KUKA KRL program: MyProgram_227().src

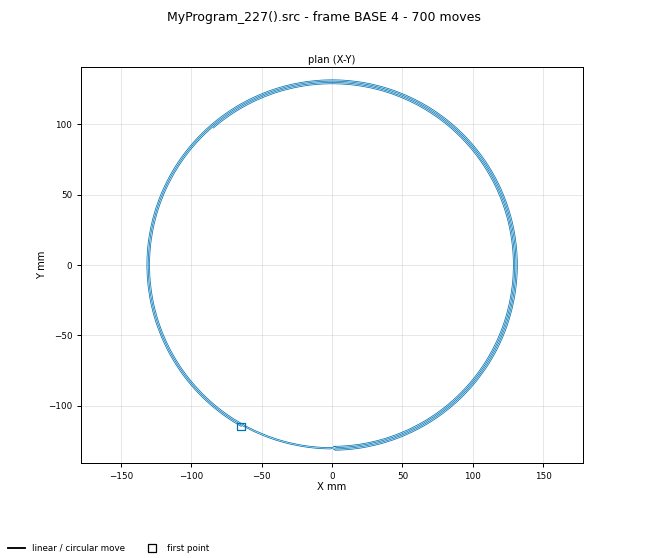
[picture p0: tool path of MyProgram_227().src in frame BASE 4, 700 of 700 moves have a stored position in this frame; points joined in program order, loops and branches not executed]
&ACCESS RVP
&REL 1
&PARAM TEMPLATE = C:\KRC\Roboter\Template\vorgabe
&PARAM EDITMASK = *
DEF MyProgram_227()
; ---- Setting reference (Base) ----
$BASE = BASE_DATA[4]

; --------------------------
; ---- Setting tool (TCP) ----
$TOOL = TOOL_DATA[3]
; --------------------------

$VEL.CP = VEL_APROX_PRINT
Startdeposition()
$VEL.CP = VEL_PRINT
LIN {X -64.5024,Y -114.7242,Z 156,A -121.3808,B 20.2003,C -0.5364,E1 20.1278,E2 209.4297} C_DIS
LIN {X -69.89,Y -111.5247,Z 156,A -124.1594,B 20.2003,C -0.5384,E1 20.1212,E2 212.2133} C_DIS
LIN {X -73.6579,Y -109.0722,Z 156,A -126.0502,B 20.2001,C -0.5441,E1 20.1168,E2 214.0953} C_DIS
LIN {X -77.2991,Y -106.5226,Z 156,A -128.0102,B 20.2001,C -0.5464,E1 20.1123,E2 216.0574} C_DIS
LIN {X -80.7887,Y -103.9011,Z 156,A -129.8858,B 20.1999,C -0.5507,E1 20.1082,E2 217.9291} C_DIS
LIN {X -84.1988,Y -101.1577,Z 156,A -131.8469,B 20.1999,C -0.552,E1 20.1039,E2 219.8956} C_DIS
LIN {X -87.3975,Y -98.4072,Z 156,A -133.6968,B 20.1998,C -0.555,E1 20.1,E2 221.746} C_DIS
LIN {X -90.6409,Y -95.4285,Z 156,A -135.5086,B 20.1996,C -0.563,E1 20.0963,E2 223.5439} C_DIS
LIN {X -93.5164,Y -92.6117,Z 156,A -137.4058,B 20.1996,C -0.561,E1 20.0926,E2 225.457} C_DIS
LIN {X -96.644,Y -89.3436,Z 156,A -139.4007,B 20.1996,C -0.5643,E1 20.0887,E2 227.4534} C_DIS
LIN {X -99.6561,Y -85.9703,Z 156,A -141.3321,B 20.1994,C -0.5702,E1 20.0852,E2 229.3787} C_DIS
LIN {X -102.7577,Y -82.2386,Z 156,A -143.5047,B 20.1994,C -0.5727,E1 20.0813,E2 231.5566} C_DIS
LIN {X -105.5327,Y -78.6451,Z 156,A -145.4674,B 20.1992,C -0.578,E1 20.078,E2 233.5158} C_DIS
LIN {X -108.1949,Y -74.9409,Z 156,A -147.3614,B 20.1989,C -0.5864,E1 20.075,E2 235.397} C_DIS
LIN {X -112.0608,Y -69.0263,Z 156,A -150.3782,B 20.1987,C -0.5965,E1 20.0705,E2 238.4037} C_DIS
LIN {X -115.078,Y -63.8693,Z 156,A -153.1743,B 20.1987,C -0.5959,E1 20.0665,E2 241.22} C_DIS
LIN {X -117.1648,Y -59.9514,Z 156,A -154.8834,B 20.1983,C -0.6097,E1 20.0643,E2 242.9005} C_DIS
LIN {X -118.6307,Y -56.9959,Z 156,A -157.3435,B 20.1993,C -0.575,E1 20.0612,E2 245.4789} C_DIS
LIN {X -121.1915,Y -51.3301,Z 156,A -159.1211,B 20.1981,C -0.6176,E1 20.0594,E2 247.1447} C_DIS
LIN {X -124.2996,Y -43.2591,Z 156,A -163.0083,B 20.1979,C -0.6237,E1 20.0555,E2 251.0416} C_DIS
LIN {X -125.3813,Y -40.0159,Z 156,A -164.4771,B 20.1977,C -0.6288,E1 20.0542,E2 252.5062} C_DIS
LIN {X -126.4456,Y -36.5168,Z 156,A -166.1537,B 20.1977,C -0.6304,E1 20.0529,E2 254.1906} C_DIS
LIN {X -127.474,Y -32.7456,Z 156,A -167.8537,B 20.1975,C -0.6355,E1 20.0517,E2 255.8881} C_DIS
LIN {X -128.2429,Y -29.5906,Z 156,A -169.2782,B 20.1974,C -0.6394,E1 20.0508,E2 257.3118} C_DIS
LIN {X -128.843,Y -26.8636,Z 156,A -170.5109,B 20.1974,C -0.6424,E1 20.0501,E2 258.5449} C_DIS
LIN {X -129.6876,Y -22.4383,Z 156,A -172.5834,B 20.1973,C -0.6443,E1 20.049,E2 260.6277} C_DIS
LIN {X -130.7797,Y -14.7915,Z 156,A -176.0889,B 20.1971,C -0.6494,E1 20.0477,E2 264.1449} C_DIS
LIN {X -131.3696,Y -7.9913,Z 156,A -178.8053,B 20.1965,C -0.6682,E1 20.0471,E2 266.827} C_DIS
LIN {X -131.6089,Y -1.0846,Z 156,A 178.2982,B 20.1961,C -0.6818,E1 20.0469,E2 269.7058} C_DIS
LIN {X -131.5118,Y 5.1452,Z 156,A 175.3937,B 20.1961,C -0.6831,E1 20.0471,E2 272.6287} C_DIS
LIN {X -131.3238,Y 8.7353,Z 156,A 173.6587,B 20.1961,C -0.6817,E1 20.0474,E2 274.3812} C_DIS
LIN {X -131.0445,Y 12.2177,Z 156,A 171.8386,B 20.1963,C -0.6754,E1 20.0478,E2 276.2337} C_DIS
LIN {X -130.5968,Y 16.3351,Z 156,A 170.3498,B 20.1957,C -0.6927,E1 20.0483,E2 277.6831} C_DIS
LIN {X -130.0557,Y 20.1816,Z 156,A 168.5773,B 20.1957,C -0.695,E1 20.049,E2 279.4623} C_DIS
LIN {X -129.1113,Y 25.5452,Z 156,A 166.2566,B 20.1953,C -0.7043,E1 20.0502,E2 281.7735} C_DIS
LIN {X -128.3484,Y 29.1287,Z 156,A 164.8371,B 20.1949,C -0.7158,E1 20.0511,E2 283.1699} C_DIS
LIN {X -127.6208,Y 32.1674,Z 156,A 163.3923,B 20.1949,C -0.7168,E1 20.052,E2 284.6224} C_DIS
LIN {X -126.7498,Y 35.4433,Z 156,A 161.9281,B 20.1947,C -0.7218,E1 20.0531,E2 286.0828} C_DIS
LIN {X -125.9037,Y 38.3411,Z 156,A 160.6577,B 20.1945,C -0.7275,E1 20.0541,E2 287.3459} C_DIS
LIN {X -124.9623,Y 41.3068,Z 156,A 159.1923,B 20.1945,C -0.7275,E1 20.0554,E2 288.8222} C_DIS
LIN {X -123.8552,Y 44.5154,Z 156,A 157.764,B 20.1943,C -0.7338,E1 20.0567,E2 290.2423} C_DIS
LIN {X -122.7696,Y 47.4281,Z 156,A 156.44,B 20.1941,C -0.7389,E1 20.058,E2 291.5607} C_DIS
LIN {X -121.5158,Y 50.5536,Z 156,A 154.8555,B 20.1941,C -0.7389,E1 20.0597,E2 293.1566} C_DIS
LIN {X -119.7827,Y 54.538,Z 156,A 152.3207,B 20.1948,C -0.7204,E1 20.0627,E2 295.763} C_DIS
LIN {X -117.5878,Y 59.1205,Z 156,A 150.668,B 20.1938,C -0.7476,E1 20.0646,E2 297.3475} C_DIS
LIN {X -115.5845,Y 62.9479,Z 156,A 148.762,B 20.1937,C -0.752,E1 20.0671,E2 299.2535} C_DIS
LIN {X -113.2985,Y 66.9761,Z 156,A 146.8963,B 20.1933,C -0.7634,E1 20.0697,E2 301.0984} C_DIS
LIN {X -111.4896,Y 69.9457,Z 156,A 145.2337,B 20.1933,C -0.7619,E1 20.0722,E2 302.7761} C_DIS
LIN {X -109.3086,Y 73.307,Z 156,A 143.4515,B 20.1933,C -0.7652,E1 20.0749,E2 304.5598} C_DIS
LIN {X -106.8382,Y 76.8632,Z 156,A 141.5225,B 20.1931,C -0.7686,E1 20.078,E2 306.4911} C_DIS
LIN {X -104.1297,Y 80.4938,Z 156,A 139.5695,B 20.1929,C -0.7744,E1 20.0813,E2 308.4389} C_DIS
LIN {X -101.2648,Y 84.0694,Z 156,A 137.5744,B 20.1927,C -0.7795,E1 20.0848,E2 310.4311} C_DIS
LIN {X -98.3299,Y 87.485,Z 156,A 135.5579,B 20.1926,C -0.7822,E1 20.0886,E2 312.4512} C_DIS
LIN {X -95.3804,Y 90.6912,Z 156,A 133.6485,B 20.1924,C -0.7863,E1 20.0922,E2 314.3593} C_DIS
LIN {X -92.0975,Y 94.0227,Z 156,A 131.6693,B 20.1922,C -0.7932,E1 20.0961,E2 316.3289} C_DIS
LIN {X -89.054,Y 96.9102,Z 156,A 129.8341,B 20.192,C -0.797,E1 20.0998,E2 318.1626} C_DIS
LIN {X -85.7986,Y 99.8039,Z 156,A 127.9139,B 20.192,C -0.8002,E1 20.1039,E2 320.083} C_DIS
LIN {X -82.5599,Y 102.4991,Z 156,A 126.0958,B 20.1917,C -0.8047,E1 20.1078,E2 321.8967} C_DIS
LIN {X -79.2878,Y 105.0507,Z 156,A 124.262,B 20.1917,C -0.8073,E1 20.1118,E2 323.7313} C_DIS
LIN {X -75.7971,Y 107.5965,Z 156,A 122.3591,B 20.1915,C -0.8102,E1 20.1162,E2 325.6344} C_DIS
LIN {X -72.1164,Y 110.0978,Z 156,A 120.4059,B 20.1915,C -0.8132,E1 20.1207,E2 327.5869} C_DIS
LIN {X -68.5529,Y 112.3513,Z 156,A 118.5367,B 20.1913,C -0.8152,E1 20.1251,E2 329.4578} C_DIS
LIN {X -64.9667,Y 114.4623,Z 156,A 116.7463,B 20.1912,C -0.8191,E1 20.1294,E2 331.2435} C_DIS
LIN {X -61.8178,Y 116.1928,Z 156,A 114.9516,B 20.1914,C -0.8127,E1 20.1339,E2 333.0633} C_DIS
LIN {X -58.9034,Y 117.6973,Z 156,A 113.719,B 20.1911,C -0.8225,E1 20.1369,E2 334.2716} C_DIS
LIN {X -55.5927,Y 119.295,Z 156,A 112.0742,B 20.1911,C -0.8231,E1 20.1411,E2 335.9197} C_DIS
LIN {X -49.197,Y 122.0712,Z 156,A 109.1849,B 20.1906,C -0.833,E1 20.1485,E2 338.7888} C_DIS
LIN {X -45.7308,Y 123.4124,Z 156,A 107.5441,B 20.1906,C -0.8341,E1 20.1528,E2 340.4307} C_DIS
LIN {X -42.1881,Y 124.6688,Z 156,A 105.8112,B 20.1906,C -0.8322,E1 20.1574,E2 342.1733} C_DIS
LIN {X -38.1859,Y 125.9512,Z 156,A 103.9702,B 20.1906,C -0.8338,E1 20.1623,E2 344.0139} C_DIS
LIN {X -33.5783,Y 127.2571,Z 156,A 101.5534,B 20.191,C -0.8227,E1 20.1689,E2 346.4674} C_DIS
LIN {X -29.7777,Y 128.2002,Z 156,A 100.0213,B 20.1907,C -0.831,E1 20.173,E2 347.9782} C_DIS
LIN {X -26.3077,Y 128.9561,Z 156,A 98.0483,B 20.1913,C -0.8153,E1 20.1785,E2 349.9994} C_DIS
LIN {X -21.1994,Y 129.8945,Z 156,A 96.3348,B 20.1904,C -0.8385,E1 20.1831,E2 351.6477} C_DIS
LIN {X -17.142,Y 130.4912,Z 156,A 94.7251,B 20.1901,C -0.8466,E1 20.1874,E2 353.2356} C_DIS
LIN {X -10.1792,Y 131.2195,Z 156,A 91.5234,B 20.1903,C -0.8417,E1 20.1964,E2 356.4535} C_DIS
LIN {X -6.3873,Y 131.4575,Z 156,A 89.89,B 20.1903,C -0.8431,E1 20.2009,E2 358.0836} C_DIS
LIN {X -2.1877,Y 131.5943,Z 156,A 88.078,B 20.1902,C -0.8442,E1 20.206,E2 359.8925} C_DIS
LIN {X 1.9611,Y 131.5981,Z 156,A 86.5669,B 20.1897,C -0.8564,E1 20.2101,E2 361.3682} C_DIS
LIN {X 5.8923,Y 131.4824,Z 156,A 84.5148,B 20.1903,C -0.8426,E1 20.2159,E2 363.4595} C_DIS
LIN {X 9.6611,Y 131.2574,Z 156,A 82.9336,B 20.1902,C -0.8451,E1 20.2203,E2 365.0327} C_DIS
LIN {X 13.7775,Y 130.8896,Z 156,A 81.0592,B 20.1902,C -0.8418,E1 20.2256,E2 366.9154} C_DIS
LIN {X 19.5443,Y 130.1544,Z 156,A 78.571,B 20.1902,C -0.8428,E1 20.2324,E2 369.3978} C_DIS
LIN {X 23.245,Y 129.5433,Z 156,A 76.9573,B 20.1902,C -0.843,E1 20.2369,E2 371.0089} C_DIS
LIN {X 28.1767,Y 128.5613,Z 156,A 74.7152,B 20.1904,C -0.8397,E1 20.243,E2 373.2569} C_DIS
LIN {X 32.0967,Y 127.6387,Z 156,A 73.1025,B 20.1902,C -0.8444,E1 20.2473,E2 374.8529} C_DIS
LIN {X 35.2064,Y 126.8161,Z 156,A 71.485,B 20.1906,C -0.8345,E1 20.2518,E2 376.4958} C_DIS
LIN {X 39.8423,Y 125.4367,Z 156,A 69.5312,B 20.1904,C -0.8392,E1 20.2569,E2 378.4316} C_DIS
LIN {X 43.2726,Y 124.2949,Z 156,A 68.0856,B 20.1902,C -0.8431,E1 20.2607,E2 379.8622} C_DIS
LIN {X 49.0275,Y 122.1395,Z 156,A 65.3591,B 20.1904,C -0.8384,E1 20.2679,E2 382.595} C_DIS
LIN {X 52.1568,Y 120.8362,Z 156,A 63.8884,B 20.1904,C -0.837,E1 20.2716,E2 384.0654} C_DIS
LIN {X 55.0772,Y 119.5334,Z 156,A 62.6797,B 20.1902,C -0.8431,E1 20.2746,E2 385.2526} C_DIS
LIN {X 57.4891,Y 118.395,Z 156,A 61.1776,B 20.1909,C -0.8272,E1 20.2785,E2 386.7954} C_DIS
LIN {X 61.0133,Y 116.6152,Z 156,A 59.6562,B 20.1906,C -0.8333,E1 20.2823,E2 388.2938} C_DIS
LIN {X 63.6126,Y 115.2201,Z 156,A 58.0731,B 20.1912,C -0.8189,E1 20.2862,E2 389.9127} C_DIS
LIN {X 68.2018,Y 112.5644,Z 156,A 55.9412,B 20.191,C -0.823,E1 20.2913,E2 392.0246} C_DIS
LIN {X 71.9413,Y 110.2124,Z 156,A 54.0685,B 20.191,C -0.8221,E1 20.2957,E2 393.8921} C_DIS
LIN {X 75.4654,Y 107.83,Z 156,A 52.1497,B 20.1913,C -0.8162,E1 20.3001,E2 395.8197} C_DIS
LIN {X 78.7314,Y 105.4685,Z 156,A 50.4574,B 20.1913,C -0.8158,E1 20.3039,E2 397.5056} C_DIS
LIN {X 82.2037,Y 102.7855,Z 156,A 48.5796,B 20.1913,C -0.8137,E1 20.308,E2 399.3806} C_DIS
LIN {X 85.4731,Y 100.0832,Z 156,A 46.7923,B 20.1914,C -0.8127,E1 20.3119,E2 401.162} C_DIS
LIN {X 88.738,Y 97.1994,Z 156,A 44.5515,B 20.1921,C -0.7942,E1 20.3166,E2 403.4449} C_DIS
LIN {X 91.3003,Y 94.7976,Z 156,A 43.2428,B 20.1919,C -0.8004,E1 20.3192,E2 404.7286} C_DIS
LIN {X 94.5144,Y 91.5928,Z 156,A 41.319,B 20.1919,C -0.7985,E1 20.3229,E2 406.6478} C_DIS
LIN {X 97.1681,Y 88.7731,Z 156,A 39.6028,B 20.1922,C -0.7934,E1 20.3262,E2 408.3689} C_DIS
LIN {X 99.6795,Y 85.9431,Z 156,A 37.9873,B 20.1922,C -0.7911,E1 20.3292,E2 409.982} C_DIS
LIN {X 102.9297,Y 82.0225,Z 156,A 35.8142,B 20.1924,C -0.7878,E1 20.333,E2 412.1518} C_DIS
LIN {X 105.4685,Y 78.7314,Z 156,A 34.1292,B 20.1924,C -0.7888,E1 20.3358,E2 413.8237} C_DIS
LIN {X 108.7981,Y 74.0628,Z 156,A 31.5163,B 20.1928,C -0.7775,E1 20.3401,E2 416.453} C_DIS
LIN {X 111.0812,Y 70.5928,Z 156,A 29.6889,B 20.193,C -0.772,E1 20.3428,E2 418.2846} C_DIS
LIN {X 113.4512,Y 66.7161,Z 156,A 27.7613,B 20.193,C -0.7691,E1 20.3456,E2 420.2082} C_DIS
LIN {X 115.67,Y 62.7911,Z 156,A 26.0407,B 20.1929,C -0.7744,E1 20.3479,E2 421.9021} C_DIS
LIN {X 118.0921,Y 58.1031,Z 156,A 23.5923,B 20.1933,C -0.7615,E1 20.351,E2 424.3711} C_DIS
LIN {X 119.7335,Y 54.6444,Z 156,A 21.83,B 20.1937,C -0.7526,E1 20.3531,E2 426.1469} C_DIS
LIN {X 121.347,Y 50.9576,Z 156,A 20.2893,B 20.1935,C -0.757,E1 20.3548,E2 427.6645} C_DIS
LIN {X 122.5599,Y 47.9675,Z 156,A 18.9069,B 20.1936,C -0.7539,E1 20.3562,E2 429.046} C_DIS
LIN {X 123.6574,Y 45.0642,Z 156,A 17.4929,B 20.1939,C -0.7472,E1 20.3576,E2 430.4693} C_DIS
LIN {X 124.7234,Y 42.0241,Z 156,A 16.1047,B 20.1939,C -0.7437,E1 20.3589,E2 431.8576} C_DIS
LIN {X 125.5276,Y 39.558,Z 156,A 14.9124,B 20.1942,C -0.7376,E1 20.3599,E2 433.059} C_DIS
LIN {X 126.8788,Y 34.9821,Z 156,A 13.0111,B 20.1942,C -0.7392,E1 20.3614,E2 434.9419} C_DIS
LIN {X 127.8142,Y 31.3943,Z 156,A 10.8889,B 20.1951,C -0.7119,E1 20.3628,E2 437.1271} C_DIS
LIN {X 128.6714,Y 27.6669,Z 156,A 9.2288,B 20.1952,C -0.707,E1 20.3638,E2 438.789} C_DIS
LIN {X 129.4575,Y 23.724,Z 156,A 7.8543,B 20.1949,C -0.7182,E1 20.3645,E2 440.1211} C_DIS
LIN {X 130.0535,Y 20.1963,Z 156,A 6.3721,B 20.1949,C -0.7168,E1 20.3652,E2 441.5965} C_DIS
LIN {X 130.8383,Y 14.2538,Z 156,A 3.5714,B 20.1955,C -0.7002,E1 20.3661,E2 444.424} C_DIS
LIN {X 131.2658,Y 9.5455,Z 156,A 1.7609,B 20.1953,C -0.7047,E1 20.3665,E2 446.2078} C_DIS
LIN {X 131.4776,Y 5.9883,Z 156,A 0.1341,B 20.1956,C -0.6965,E1 20.3668,E2 447.8461} C_DIS
LIN {X 131.5938,Y 2.2195,Z 156,A -1.4535,B 20.1956,C -0.6937,E1 20.3668,E2 449.4297} C_DIS
LIN {X 131.5982,Y -1.9522,Z 156,A -3.2301,B 20.1958,C -0.6897,E1 20.3668,E2 451.2044} C_DIS
LIN {X 131.4915,Y -5.6661,Z 156,A -4.9406,B 20.1961,C -0.6805,E1 20.3667,E2 452.9287} C_DIS
LIN {X 131.2776,Y -9.3838,Z 156,A -6.319,B 20.1959,C -0.6862,E1 20.3664,E2 454.2803} C_DIS
LIN {X 130.6782,Y -15.6533,Z 156,A -9.1651,B 20.1964,C -0.6728,E1 20.3656,E2 457.1434} C_DIS
LIN {X 130.144,Y -19.6118,Z 156,A -10.7532,B 20.1964,C -0.6741,E1 20.365,E2 458.7162} C_DIS
LIN {X 129.3929,Y -24.0765,Z 156,A -12.882,B 20.1967,C -0.6608,E1 20.364,E2 460.8672} C_DIS
LIN {X 127.674,Y -31.9578,Z 156,A -17.4583,B 20.1985,C -0.603,E1 20.361,E2 465.5762} C_DIS
LIN {X 125.5974,Y -39.3394,Z 156,A -19.7302,B 20.1974,C -0.6396,E1 20.3592,E2 467.7264} C_DIS
LIN {X 124.5474,Y -42.5443,Z 156,A -21.0624,B 20.1974,C -0.6412,E1 20.3581,E2 469.0446} C_DIS
LIN {X 123.3126,Y -45.9974,Z 156,A -23.4632,B 20.1985,C -0.6009,E1 20.3556,E2 471.5444} C_DIS
LIN {X 121.1237,Y -51.4912,Z 156,A -25.2866,B 20.1978,C -0.6263,E1 20.3538,E2 473.282} C_DIS
LIN {X 119.6012,Y -54.9305,Z 156,A -26.6816,B 20.1976,C -0.6323,E1 20.3522,E2 474.6503} C_DIS
LIN {X 118.8149,Y -56.6104,Z 156,A -28.0066,B 20.1984,C -0.607,E1 20.3505,E2 476.039} C_DIS
LIN {X 117.2458,Y -59.7924,Z 156,A -29.0782,B 20.1979,C -0.6234,E1 20.3493,E2 477.0561} C_DIS
LIN {X 115.7121,Y -62.7141,Z 156,A -30.7188,B 20.1983,C -0.6102,E1 20.3471,E2 478.7237} C_DIS
LIN {X 113.701,Y -66.2907,Z 156,A -32.4644,B 20.1983,C -0.6069,E1 20.3446,E2 480.4673} C_DIS
LIN {X 111.5286,Y -69.8839,Z 156,A -34.2997,B 20.1985,C -0.6015,E1 20.3419,E2 482.3064} C_DIS
LIN {X 109.1962,Y -73.4747,Z 156,A -36.1344,B 20.1986,C -0.5977,E1 20.3391,E2 484.1405} C_DIS
LIN {X 104.0032,Y -80.6569,Z 156,A -40.1372,B 20.1991,C -0.5811,E1 20.3325,E2 488.1666} C_DIS
LIN {X 101.5007,Y -83.7846,Z 156,A -42.1923,B 20.1996,C -0.563,E1 20.3288,E2 490.2619} C_DIS
LIN {X 98.4389,Y -87.3616,Z 156,A -43.6096,B 20.199,C -0.5856,E1 20.3263,E2 491.6061} C_DIS
LIN {X 93.3518,Y -92.7774,Z 156,A -46.8661,B 20.1992,C -0.5768,E1 20.32,E2 494.8701} C_DIS
LIN {X 88.3975,Y -97.5095,Z 156,A -50.1148,B 20.1997,C -0.5583,E1 20.3133,E2 498.1552} C_DIS
LIN {X 83.9468,Y -101.3663,Z 156,A -52.4094,B 20.1995,C -0.5644,E1 20.3085,E2 500.4208} C_DIS
LIN {X 78.3102,Y -105.7821,Z 156,A -55.623,B 20.1998,C -0.5537,E1 20.3013,E2 503.6504} C_DIS
LIN {X 74.6594,Y -108.3892,Z 156,A -57.5017,B 20.1998,C -0.5531,E1 20.297,E2 505.5226} C_DIS
LIN {X 71.3089,Y -110.6229,Z 156,A -59.4292,B 20.2001,C -0.5422,E1 20.2925,E2 507.4733} C_DIS
LIN {X 66.739,Y -113.4378,Z 156,A -61.5372,B 20.2,C -0.5479,E1 20.2875,E2 509.5566} C_DIS
LIN {X 63.2524,Y -115.4184,Z 156,A -63.1592,B 20.2,C -0.5503,E1 20.2836,E2 511.1658} C_DIS
LIN {X 57.3027,Y -118.4841,Z 156,A -66.1346,B 20.2001,C -0.5429,E1 20.2762,E2 514.1521} C_DIS
LIN {X 53.848,Y -120.0921,Z 156,A -67.7383,B 20.2001,C -0.5429,E1 20.2721,E2 515.7509} C_DIS
LIN {X 51.3763,Y -121.1722,Z 156,A -69.004,B 20.2003,C -0.5372,E1 20.2688,E2 517.0289} C_DIS
LIN {X 47.3272,Y -122.8088,Z 156,A -70.9608,B 20.2003,C -0.5323,E1 20.2637,E2 518.9944} C_DIS
LIN {X 43.1661,Y -124.3319,Z 156,A -72.7643,B 20.2003,C -0.5353,E1 20.259,E2 520.7846} C_DIS
LIN {X 37.2335,Y -126.2358,Z 156,A -75.7877,B 20.2007,C -0.519,E1 20.2508,E2 523.848} C_DIS
LIN {X 34.0665,Y -127.1269,Z 156,A -76.89,B 20.2004,C -0.5316,E1 20.248,E2 524.9119} C_DIS
LIN {X 30.9231,Y -127.9278,Z 156,A -78.2553,B 20.2004,C -0.5322,E1 20.2443,E2 526.2727} C_DIS
LIN {X 24.2335,Y -129.3629,Z 156,A -81.2641,B 20.2004,C -0.5284,E1 20.2361,E2 529.2877} C_DIS
LIN {X 21.8709,Y -129.7825,Z 156,A -82.7006,B 20.2009,C -0.5112,E1 20.232,E2 530.772} C_DIS
LIN {X 18.2798,Y -130.3371,Z 156,A -84.0182,B 20.2007,C -0.5213,E1 20.2284,E2 532.0591} C_DIS
LIN {X 14.3884,Y -130.8238,Z 156,A -85.6588,B 20.2007,C -0.5231,E1 20.2239,E2 533.6928} C_DIS
LIN {X 10.3975,Y -131.2028,Z 156,A -87.4427,B 20.2007,C -0.5206,E1 20.2189,E2 535.4825} C_DIS
LIN {X 6.4754,Y -131.4531,Z 156,A -89.1069,B 20.2007,C -0.522,E1 20.2143,E2 537.142} C_DIS
LIN {X 2.2514,Y -131.5932,Z 156,A -90.9121,B 20.2007,C -0.5229,E1 20.2092,E2 538.944} C_DIS
LIN {X 2.2514,Y -131.5932,Z 156,A -90.9121,B 20.2007,C -0.5229,E1 20.2092,E2 538.944} C_DIS
Enddeposition()
LIN {X 0.9052,Y -130.6755,Z 156,A -91.1331,B 18.9222,C -0.3682,E1 18.9261,E2 539.5117} C_DIS
Startdeposition()
$VEL.CP = VEL_PRINT
LIN {X 5.0067,Y -130.5828,Z 156,A -88.6405,B 18.9216,C -0.3957,E1 18.9333,E2 536.9351} C_DIS
LIN {X 8.8903,Y -130.3774,Z 156,A -86.9352,B 18.9216,C -0.3963,E1 18.9381,E2 535.2288} C_DIS
LIN {X 12.4269,Y -130.0864,Z 156,A -85.3683,B 18.9216,C -0.3975,E1 18.9424,E2 533.6595} C_DIS
LIN {X 16.5957,Y -129.621,Z 156,A -83.5782,B 18.9216,C -0.3965,E1 18.9474,E2 531.8742} C_DIS
LIN {X 22.9346,Y -128.6502,Z 156,A -80.8451,B 18.9216,C -0.3953,E1 18.9549,E2 529.1486} C_DIS
LIN {X 30.7927,Y -126.9988,Z 156,A -77.431,B 18.9216,C -0.3939,E1 18.9642,E2 525.7449} C_DIS
LIN {X 36.1822,Y -125.5707,Z 156,A -74.4087,B 18.9211,C -0.4195,E1 18.9725,E2 522.6506} C_DIS
LIN {X 39.6405,Y -124.521,Z 156,A -73.143,B 18.9214,C -0.4084,E1 18.9758,E2 521.4221} C_DIS
LIN {X 43.8451,Y -123.1043,Z 156,A -71.2127,B 18.9214,C -0.4101,E1 18.9809,E2 519.4919} C_DIS
LIN {X 47.3236,Y -121.8083,Z 156,A -69.6873,B 18.9214,C -0.4081,E1 18.9848,E2 517.9772} C_DIS
LIN {X 49.9928,Y -120.738,Z 156,A -68.221,B 18.9212,C -0.4181,E1 18.9887,E2 516.4847} C_DIS
LIN {X 54.5977,Y -118.7264,Z 156,A -66.431,B 18.9214,C -0.4045,E1 18.9931,E2 514.7424} C_DIS
LIN {X 59.6854,Y -116.2524,Z 156,A -63.7114,B 18.9212,C -0.418,E1 19,E2 511.9913} C_DIS
LIN {X 63.512,Y -114.2085,Z 156,A -61.7575,B 18.921,C -0.4232,E1 19.0048,E2 510.0291} C_DIS
LIN {X 67.1764,Y -112.0924,Z 156,A -59.6628,B 18.9208,C -0.4362,E1 19.01,E2 507.9031} C_DIS
LIN {X 70.0987,Y -110.2888,Z 156,A -58.3792,B 18.9209,C -0.4299,E1 19.0129,E2 506.6447} C_DIS
LIN {X 73.714,Y -107.9056,Z 156,A -56.5242,B 18.9209,C -0.4317,E1 19.0172,E2 504.7926} C_DIS
LIN {X 77.2438,Y -105.4073,Z 156,A -54.895,B 18.921,C -0.4244,E1 19.0208,E2 503.1934} C_DIS
LIN {X 82.5021,Y -101.3447,Z 156,A -51.7147,B 18.9206,C -0.4414,E1 19.0279,E2 499.9771} C_DIS
LIN {X 85.9475,Y -98.4394,Z 156,A -49.7809,B 18.9206,C -0.4439,E1 19.032,E2 498.0458} C_DIS
LIN {X 88.9068,Y -95.775,Z 156,A -47.5299,B 18.92,C -0.4688,E1 19.0368,E2 495.7309} C_DIS
LIN {X 92.363,Y -92.4472,Z 156,A -45.9363,B 18.9204,C -0.4525,E1 19.0398,E2 494.1966} C_DIS
LIN {X 96.4676,Y -88.1557,Z 156,A -43.4115,B 18.9204,C -0.4554,E1 19.0446,E2 491.6777} C_DIS
LIN {X 100.555,Y -83.4625,Z 156,A -40.6492,B 18.9201,C -0.4636,E1 19.0497,E2 488.9074} C_DIS
LIN {X 103.3035,Y -80.0355,Z 156,A -37.9705,B 18.9192,C -0.5001,E1 19.0544,E2 486.134} C_DIS
LIN {X 106.9356,Y -75.1141,Z 156,A -36.0855,B 18.9199,C -0.4736,E1 19.0573,E2 484.3425} C_DIS
LIN {X 109.2436,Y -71.7158,Z 156,A -34.2865,B 18.9198,C -0.4784,E1 19.0601,E2 482.541} C_DIS
LIN {X 111.4646,Y -68.2126,Z 156,A -32.4871,B 18.9197,C -0.4826,E1 19.0627,E2 480.7413} C_DIS
LIN {X 113.7219,Y -64.38,Z 156,A -30.5032,B 18.9195,C -0.4894,E1 19.0655,E2 478.7503} C_DIS
LIN {X 115.7765,Y -60.6019,Z 156,A -28.7571,B 18.9195,C -0.489,E1 19.0678,E2 477.0182} C_DIS
LIN {X 118.4529,Y -55.1891,Z 156,A -26.1109,B 18.9193,C -0.4965,E1 19.071,E2 474.3682} C_DIS
LIN {X 120.2831,Y -51.0789,Z 156,A -23.2694,B 18.9182,C -0.539,E1 19.0743,E2 471.4175} C_DIS
LIN {X 122.6579,Y -45.083,Z 156,A -21.2294,B 18.9189,C -0.514,E1 19.0762,E2 469.4695} C_DIS
LIN {X 123.9393,Y -41.4233,Z 156,A -19.8022,B 18.919,C -0.5077,E1 19.0774,E2 468.0727} C_DIS
LIN {X 124.9991,Y -38.106,Z 156,A -17.4959,B 18.918,C -0.5452,E1 19.0794,E2 465.6693} C_DIS
LIN {X 126.4376,Y -33.0275,Z 156,A -15.7772,B 18.9185,C -0.527,E1 19.0806,E2 464.0197} C_DIS
LIN {X 127.2358,Y -29.8065,Z 156,A -14.0493,B 18.9181,C -0.543,E1 19.0817,E2 462.2564} C_DIS
LIN {X 127.9985,Y -26.3301,Z 156,A -12.8924,B 18.9184,C -0.5308,E1 19.0824,E2 461.146} C_DIS
LIN {X 129.2709,Y -19.1403,Z 156,A -9.6278,B 18.9181,C -0.5434,E1 19.0839,E2 457.8691} C_DIS
LIN {X 130.1332,Y -11.925,Z 156,A -6.6336,B 18.9181,C -0.5452,E1 19.0848,E2 454.8932} C_DIS
LIN {X 130.4338,Y -7.9966,Z 156,A -4.8089,B 18.9178,C -0.5547,E1 19.0852,E2 453.0543} C_DIS
LIN {X 130.6217,Y -3.8656,Z 156,A -3.0252,B 18.9177,C -0.5591,E1 19.0854,E2 451.2714} C_DIS
LIN {X 130.6786,Y -0.3496,Z 156,A -1.4346,B 18.9175,C -0.566,E1 19.0854,E2 449.6726} C_DIS
LIN {X 130.6276,Y 3.6539,Z 156,A 0.2672,B 18.9174,C -0.5692,E1 19.0853,E2 447.9747} C_DIS
LIN {X 130.4451,Y 7.8125,Z 156,A 2.0701,B 18.9172,C -0.5739,E1 19.085,E2 446.1719} C_DIS
LIN {X 130.2398,Y 10.704,Z 156,A 3.7221,B 18.9166,C -0.5939,E1 19.0847,E2 444.4721} C_DIS
LIN {X 129.8527,Y 14.6857,Z 156,A 5.7568,B 18.9161,C -0.6112,E1 19.084,E2 442.4008} C_DIS
LIN {X 129.1444,Y 19.9649,Z 156,A 7.3594,B 18.9168,C -0.5874,E1 19.0834,E2 440.8838} C_DIS
LIN {X 128.7001,Y 22.6556,Z 156,A 8.9728,B 18.9162,C -0.6086,E1 19.0826,E2 439.2184} C_DIS
LIN {X 127.9596,Y 26.5197,Z 156,A 10.3455,B 18.9165,C -0.599,E1 19.0818,E2 437.8859} C_DIS
LIN {X 126.4118,Y 33.1241,Z 156,A 13.1417,B 18.9165,C -0.6004,E1 19.08,E2 435.1073} C_DIS
LIN {X 125.5707,Y 36.1822,Z 156,A 14.4641,B 18.9164,C -0.6017,E1 19.079,E2 433.7913} C_DIS
LIN {X 124.5388,Y 39.5847,Z 156,A 16.1018,B 18.9161,C -0.6096,E1 19.0776,E2 432.1422} C_DIS
LIN {X 123.4248,Y 42.932,Z 156,A 17.6503,B 18.9161,C -0.6141,E1 19.0762,E2 430.5916} C_DIS
LIN {X 122.0893,Y 46.6009,Z 156,A 19.4974,B 18.9157,C -0.6246,E1 19.0744,E2 428.7263} C_DIS
LIN {X 120.6642,Y 50.1697,Z 156,A 21.0297,B 18.9157,C -0.6231,E1 19.0728,E2 427.2102} C_DIS
LIN {X 119.3571,Y 53.2042,Z 156,A 22.4643,B 18.9157,C -0.6265,E1 19.0712,E2 425.7756} C_DIS
LIN {X 118.1494,Y 55.8373,Z 156,A 24.2239,B 18.9148,C -0.6504,E1 19.069,E2 423.9558} C_DIS
LIN {X 116.283,Y 59.6254,Z 156,A 25.6936,B 18.9152,C -0.6395,E1 19.0672,E2 422.5301} C_DIS
LIN {X 114.2241,Y 63.4837,Z 156,A 27.5025,B 18.9152,C -0.6401,E1 19.0648,E2 420.7323} C_DIS
LIN {X 112.2691,Y 66.88,Z 156,A 29.2673,B 18.915,C -0.6465,E1 19.0623,E2 418.9601} C_DIS
LIN {X 109.8864,Y 70.7275,Z 156,A 31.2167,B 18.9148,C -0.6502,E1 19.0594,E2 417.013} C_DIS
LIN {X 106.5969,Y 75.5933,Z 156,A 33.8812,B 18.9145,C -0.6602,E1 19.0552,E2 414.3354} C_DIS
LIN {X 103.5846,Y 79.6721,Z 156,A 36.021,B 18.9145,C -0.6621,E1 19.0516,E2 412.2036} C_DIS
LIN {X 101.568,Y 82.227,Z 156,A 37.6685,B 18.914,C -0.6745,E1 19.0487,E2 410.5286} C_DIS
LIN {X 99.3548,Y 84.8883,Z 156,A 38.9348,B 18.9143,C -0.6677,E1 19.0464,E2 409.2912} C_DIS
LIN {X 96.4696,Y 88.1535,Z 156,A 40.9204,B 18.914,C -0.675,E1 19.0427,E2 407.2952} C_DIS
LIN {X 93.0425,Y 91.7634,Z 156,A 43.0169,B 18.914,C -0.6761,E1 19.0386,E2 405.2073} C_DIS
LIN {X 90.2107,Y 94.548,Z 156,A 45.1123,B 18.9133,C -0.6942,E1 19.0343,E2 403.0684} C_DIS
LIN {X 87.1704,Y 97.3582,Z 156,A 46.5257,B 18.9138,C -0.6814,E1 19.0315,E2 401.702} C_DIS
LIN {X 83.8438,Y 100.2374,Z 156,A 48.1912,B 18.914,C -0.6744,E1 19.028,E2 400.0667} C_DIS
LIN {X 81.1814,Y 102.4057,Z 156,A 49.9517,B 18.9136,C -0.6875,E1 19.0241,E2 398.2751} C_DIS
LIN {X 77.6585,Y 105.1027,Z 156,A 51.8796,B 18.9135,C -0.6902,E1 19.0198,E2 396.3483} C_DIS
LIN {X 74.1762,Y 107.5884,Z 156,A 53.7702,B 18.9133,C -0.6939,E1 19.0155,E2 394.4551} C_DIS
LIN {X 70.5676,Y 109.9887,Z 156,A 55.6191,B 18.9133,C -0.6949,E1 19.0112,E2 392.6116} C_DIS
LIN {X 67.002,Y 112.1964,Z 156,A 57.6077,B 18.913,C -0.7036,E1 19.0064,E2 390.6046} C_DIS
LIN {X 62.6853,Y 114.6641,Z 156,A 59.6409,B 18.9131,C -0.7008,E1 19.0015,E2 388.5882} C_DIS
LIN {X 59.6447,Y 116.2732,Z 156,A 61.0946,B 18.9131,C -0.7006,E1 18.9979,E2 387.1405} C_DIS
LIN {X 56.4944,Y 117.8354,Z 156,A 62.65,B 18.9131,C -0.7031,E1 18.994,E2 385.5832} C_DIS
LIN {X 53.2541,Y 119.3348,Z 156,A 64.137,B 18.9131,C -0.7018,E1 18.9902,E2 384.1052} C_DIS
LIN {X 49.6887,Y 120.865,Z 156,A 66.3099,B 18.9123,C -0.7223,E1 18.9845,E2 381.8763} C_DIS
LIN {X 46.0462,Y 122.2971,Z 156,A 67.7189,B 18.9127,C -0.7118,E1 18.9809,E2 380.5035} C_DIS
LIN {X 41.7478,Y 123.8312,Z 156,A 69.4428,B 18.913,C -0.7027,E1 18.9764,E2 378.8124} C_DIS
LIN {X 38.3204,Y 124.9335,Z 156,A 71.0438,B 18.913,C -0.7049,E1 18.9721,E2 377.2088} C_DIS
LIN {X 34.1847,Y 126.129,Z 156,A 73.0821,B 18.9127,C -0.7121,E1 18.9666,E2 375.1528} C_DIS
LIN {X 30.8031,Y 126.9962,Z 156,A 74.448,B 18.9129,C -0.7067,E1 18.963,E2 373.8065} C_DIS
LIN {X 28.3775,Y 127.5622,Z 156,A 75.6088,B 18.9128,C -0.7099,E1 18.9598,E2 372.6379} C_DIS
LIN {X 25.3252,Y 128.2029,Z 156,A 77.2464,B 18.9124,C -0.7211,E1 18.9552,E2 370.9687} C_DIS
LIN {X 20.3201,Y 129.0894,Z 156,A 79.0258,B 18.913,C -0.7046,E1 18.9505,E2 369.2426} C_DIS
LIN {X 15.0946,Y 129.8044,Z 156,A 81.6623,B 18.9125,C -0.7176,E1 18.9431,E2 366.5688} C_DIS
LIN {X 10.7567,Y 130.2354,Z 156,A 83.5277,B 18.9125,C -0.7161,E1 18.9379,E2 364.7095} C_DIS
LIN {X 6.0464,Y 130.5397,Z 156,A 85.726,B 18.9124,C -0.7211,E1 18.9317,E2 362.4969} C_DIS
LIN {X 1.0722,Y 130.6748,Z 156,A 87.728,B 18.9126,C -0.7141,E1 18.9262,E2 360.517} C_DIS
LIN {X -2.6987,Y 130.6519,Z 156,A 89.4744,B 18.9126,C -0.7173,E1 18.9213,E2 358.7606} C_DIS
LIN {X -6.6282,Y 130.5105,Z 156,A 91.1061,B 18.9126,C -0.7134,E1 18.9168,E2 357.1407} C_DIS
LIN {X -10.1444,Y 130.2858,Z 156,A 92.5822,B 18.9128,C -0.7102,E1 18.9127,E2 355.6735} C_DIS
LIN {X -14.2577,Y 129.8988,Z 156,A 95.0223,B 18.9119,C -0.7332,E1 18.9057,E2 353.1605} C_DIS
LIN {X -18.8877,Y 129.307,Z 156,A 96.4618,B 18.9128,C -0.7091,E1 18.9019,E2 351.794} C_DIS
LIN {X -23.7539,Y 128.5023,Z 156,A 99.1125,B 18.9122,C -0.726,E1 18.8945,E2 349.0875} C_DIS
LIN {X -27.621,Y 127.726,Z 156,A 100.0405,B 18.9133,C -0.6947,E1 18.8922,E2 348.2547} C_DIS
LIN {X -32.8223,Y 126.491,Z 156,A 102.8529,B 18.9128,C -0.71,E1 18.8844,E2 345.3898} C_DIS
LIN {X -36.5112,Y 125.4743,Z 156,A 104.4057,B 18.913,C -0.7037,E1 18.8803,E2 343.853} C_DIS
LIN {X -39.3549,Y 124.6122,Z 156,A 105.9179,B 18.9128,C -0.7101,E1 18.8762,E2 342.3175} C_DIS
LIN {X -44.1597,Y 122.9909,Z 156,A 107.9458,B 18.9131,C -0.7003,E1 18.8709,E2 340.3146} C_DIS
LIN {X -47.2076,Y 121.8534,Z 156,A 109.3923,B 18.9131,C -0.6993,E1 18.8671,E2 338.8671} C_DIS
LIN {X -53.6882,Y 119.1407,Z 156,A 112.572,B 18.9131,C -0.6988,E1 18.859,E2 335.679} C_DIS
LIN {X -57.5344,Y 117.3314,Z 156,A 114.3255,B 18.9134,C -0.692,E1 18.8546,E2 333.9404} C_DIS
LIN {X -59.8953,Y 116.1456,Z 156,A 115.5715,B 18.9134,C -0.6934,E1 18.8515,E2 332.6855} C_DIS
LIN {X -63.6262,Y 114.1453,Z 156,A 117.5084,B 18.9134,C -0.6934,E1 18.8467,E2 330.7412} C_DIS
LIN {X -67.241,Y 112.054,Z 156,A 119.3131,B 18.9135,C -0.6893,E1 18.8424,E2 328.9418} C_DIS
LIN {X -70.7534,Y 109.8698,Z 156,A 121.1204,B 18.9136,C -0.6858,E1 18.8381,E2 327.1374} C_DIS
LIN {X -74.269,Y 107.5247,Z 156,A 123.0414,B 18.9136,C -0.6849,E1 18.8337,E2 325.2107} C_DIS
LIN {X -77.9208,Y 104.9079,Z 156,A 124.9598,B 18.9139,C -0.6792,E1 18.8294,E2 323.3007} C_DIS
LIN {X -81.211,Y 102.3822,Z 156,A 126.8291,B 18.9139,C -0.6773,E1 18.8252,E2 321.4278} C_DIS
LIN {X -84.7542,Y 99.4688,Z 156,A 128.8188,B 18.9141,C -0.6723,E1 18.821,E2 319.4432} C_DIS
LIN {X -88.0982,Y 96.5202,Z 156,A 130.8314,B 18.9141,C -0.6701,E1 18.8168,E2 317.4265} C_DIS
LIN {X -91.2647,Y 93.5316,Z 156,A 132.7523,B 18.9143,C -0.6662,E1 18.8129,E2 315.5068} C_DIS
LIN {X -94.4144,Y 90.3505,Z 156,A 134.7029,B 18.9145,C -0.6612,E1 18.8091,E2 313.5603} C_DIS
LIN {X -97.5338,Y 86.9742,Z 156,A 136.7338,B 18.9146,C -0.6569,E1 18.8053,E2 311.5304} C_DIS
LIN {X -100.3339,Y 83.7288,Z 156,A 138.6484,B 18.9147,C -0.6536,E1 18.8019,E2 309.6145} C_DIS
LIN {X -103.0946,Y 80.305,Z 156,A 140.5975,B 18.9149,C -0.6494,E1 18.7985,E2 307.6657} C_DIS
LIN {X -105.7576,Y 76.7635,Z 156,A 142.522,B 18.9151,C -0.6438,E1 18.7953,E2 305.7461} C_DIS
LIN {X -108.1947,Y 73.2885,Z 156,A 144.3672,B 18.9152,C -0.6383,E1 18.7924,E2 303.9056} C_DIS
LIN {X -110.5975,Y 69.6097,Z 156,A 146.1907,B 18.9155,C -0.6294,E1 18.7897,E2 302.097} C_DIS
LIN {X -111.8519,Y 67.5754,Z 156,A 147.4264,B 18.9155,C -0.6332,E1 18.7879,E2 300.8409} C_DIS
LIN {X -113.8711,Y 64.1146,Z 156,A 149.1417,B 18.9156,C -0.6269,E1 18.7855,E2 299.1331} C_DIS
LIN {X -115.4723,Y 61.1812,Z 156,A 150.6359,B 18.9157,C -0.6238,E1 18.7835,E2 297.6377} C_DIS
LIN {X -117.7738,Y 56.6234,Z 156,A 153.0163,B 18.9157,C -0.6224,E1 18.7806,E2 295.2441} C_DIS
LIN {X -119.8662,Y 52.0474,Z 156,A 155.0331,B 18.9162,C -0.6093,E1 18.7783,E2 293.2529} C_DIS
LIN {X -121.0455,Y 49.2439,Z 156,A 156.3772,B 18.9162,C -0.6058,E1 18.7769,E2 291.9096} C_DIS
LIN {X -122.1993,Y 46.3076,Z 156,A 157.8216,B 18.9163,C -0.6038,E1 18.7754,E2 290.4602} C_DIS
LIN {X -123.4289,Y 42.9201,Z 156,A 159.4102,B 18.9165,C -0.5994,E1 18.7739,E2 288.873} C_DIS
LIN {X -124.757,Y 38.8969,Z 156,A 161.3772,B 18.9165,C -0.5977,E1 18.7723,E2 286.8961} C_DIS
LIN {X -125.8466,Y 35.2059,Z 156,A 162.919,B 18.9168,C -0.5875,E1 18.7711,E2 285.3739} C_DIS
LIN {X -126.6192,Y 32.3181,Z 156,A 164.3015,B 18.9168,C -0.586,E1 18.7701,E2 283.985} C_DIS
LIN {X -127.5791,Y 28.3016,Z 156,A 166.1846,B 18.917,C -0.583,E1 18.7689,E2 282.0963} C_DIS
LIN {X -128.3693,Y 24.4577,Z 156,A 168.1126,B 18.9169,C -0.585,E1 18.7679,E2 280.1464} C_DIS
LIN {X -128.934,Y 21.2822,Z 156,A 169.2439,B 18.9173,C -0.5706,E1 18.7674,E2 279.0506} C_DIS
LIN {X -129.5408,Y 17.2083,Z 156,A 171.0963,B 18.9174,C -0.5667,E1 18.7667,E2 277.1955} C_DIS
LIN {X -129.9422,Y 13.8539,Z 156,A 172.7525,B 18.9174,C -0.5682,E1 18.7661,E2 275.5209} C_DIS
LIN {X -130.53,Y 6.2402,Z 156,A 175.7288,B 18.9181,C -0.5447,E1 18.7656,E2 272.5933} C_DIS
LIN {X -130.6796,Y -0.1352,Z 156,A 178.7652,B 18.9181,C -0.5443,E1 18.7654,E2 269.533} C_DIS
LIN {X -130.4958,Y -6.9193,Z 156,A -178.1647,B 18.9182,C -0.5384,E1 18.7657,E2 266.4563} C_DIS
LIN {X -130.2057,Y -11.1087,Z 156,A -175.8236,B 18.9179,C -0.5504,E1 18.7663,E2 264.0587} C_DIS
LIN {X -129.7403,Y -15.6318,Z 156,A -174.051,B 18.9183,C -0.5364,E1 18.7668,E2 262.3151} C_DIS
LIN {X -129.2879,Y -19.0214,Z 156,A -172.7425,B 18.9186,C -0.5251,E1 18.7673,E2 261.0313} C_DIS
LIN {X -128.6303,Y -23.0459,Z 156,A -171.0898,B 18.9189,C -0.5149,E1 18.7681,E2 259.3969} C_DIS
LIN {X -127.7923,Y -27.3141,Z 156,A -169.087,B 18.9189,C -0.5125,E1 18.7692,E2 257.3853} C_DIS
LIN {X -126.956,Y -30.9701,Z 156,A -167.3864,B 18.9189,C -0.5096,E1 18.7703,E2 255.6803} C_DIS
LIN {X -125.901,Y -35.0115,Z 156,A -165.6071,B 18.9192,C -0.5023,E1 18.7716,E2 253.9095} C_DIS
LIN {X -124.8988,Y -38.4336,Z 156,A -164.0363,B 18.9192,C -0.498,E1 18.7729,E2 252.3397} C_DIS
LIN {X -123.6872,Y -42.1751,Z 156,A -162.3905,B 18.9195,C -0.4902,E1 18.7743,E2 250.7054} C_DIS
LIN {X -121.4202,Y -48.3144,Z 156,A -159.3805,B 18.9195,C -0.4869,E1 18.7773,E2 247.6824} C_DIS
LIN {X -120.0545,Y -51.6118,Z 156,A -157.8508,B 18.9197,C -0.4813,E1 18.7789,E2 246.1586} C_DIS
LIN {X -117.4879,Y -57.2173,Z 156,A -155.0368,B 18.9197,C -0.4778,E1 18.7823,E2 243.3346} C_DIS
LIN {X -115.832,Y -60.4964,Z 156,A -153.5045,B 18.92,C -0.4707,E1 18.7842,E2 241.8133} C_DIS
LIN {X -113.9251,Y -64.0185,Z 156,A -151.2437,B 18.9196,C -0.4842,E1 18.7874,E2 239.4944} C_DIS
LIN {X -111.8202,Y -67.6279,Z 156,A -149.8455,B 18.9201,C -0.4638,E1 18.7893,E2 238.1497} C_DIS
LIN {X -110.4318,Y -69.8722,Z 156,A -148.1472,B 18.9197,C -0.4804,E1 18.792,E2 236.388} C_DIS
LIN {X -107.8904,Y -73.7361,Z 156,A -146.5644,B 18.9202,C -0.4592,E1 18.7944,E2 234.8603} C_DIS
LIN {X -105.2042,Y -77.5203,Z 156,A -144.5573,B 18.9204,C -0.4533,E1 18.7976,E2 232.8583} C_DIS
LIN {X -102.5544,Y -80.9938,Z 156,A -142.5877,B 18.9204,C -0.4508,E1 18.801,E2 230.884} C_DIS
LIN {X -99.7987,Y -84.3661,Z 156,A -140.6508,B 18.9205,C -0.4474,E1 18.8045,E2 228.9453} C_DIS
LIN {X -96.7013,Y -87.8986,Z 156,A -138.6686,B 18.9207,C -0.44,E1 18.8081,E2 226.9739} C_DIS
LIN {X -93.8134,Y -90.9744,Z 156,A -136.6271,B 18.9207,C -0.4431,E1 18.8121,E2 224.9108} C_DIS
LIN {X -90.1771,Y -94.5801,Z 156,A -134.5046,B 18.9208,C -0.434,E1 18.8163,E2 222.8045} C_DIS
LIN {X -86.9349,Y -97.5691,Z 156,A -132.5573,B 18.9208,C -0.4307,E1 18.8204,E2 220.8568} C_DIS
LIN {X -83.8259,Y -100.2525,Z 156,A -130.7559,B 18.921,C -0.4274,E1 18.8242,E2 219.0564} C_DIS
LIN {X -80.3949,Y -103.0249,Z 156,A -128.7735,B 18.921,C -0.4257,E1 18.8285,E2 217.0691} C_DIS
LIN {X -76.8789,Y -105.6739,Z 156,A -126.9039,B 18.9211,C -0.4201,E1 18.8327,E2 215.2078} C_DIS
LIN {X -74.364,Y -107.4584,Z 156,A -125.4751,B 18.9211,C -0.4208,E1 18.836,E2 213.7703} C_DIS
LIN {X -70.7453,Y -109.875,Z 156,A -123.45,B 18.9211,C -0.4222,E1 18.8408,E2 211.732} C_DIS
LIN {X -66.0464,Y -112.7617,Z 156,A -121.2299,B 18.9213,C -0.4113,E1 18.846,E2 209.5363} C_DIS
LIN {X -62.597,Y -114.7123,Z 156,A -119.4913,B 18.9213,C -0.4089,E1 18.8503,E2 207.7981} C_DIS
LIN {X -59.4793,Y -116.3574,Z 156,A -117.9933,B 18.9214,C -0.4052,E1 18.854,E2 206.3061} C_DIS
LIN {X -56.678,Y -117.7478,Z 156,A -116.5686,B 18.9214,C -0.4056,E1 18.8576,E2 204.8753} C_DIS
LIN {X -52.8614,Y -119.5105,Z 156,A -114.2505,B 18.9211,C -0.4215,E1 18.8636,E2 202.5003} C_DIS
LIN {X -49.09,Y -121.1075,Z 156,A -112.8194,B 18.9214,C -0.4058,E1 18.8672,E2 201.1133} C_DIS
LIN {X -44.7606,Y -122.7742,Z 156,A -111.0181,B 18.9216,C -0.3951,E1 18.8718,E2 199.34} C_DIS
LIN {X -41.4561,Y -123.9284,Z 156,A -109.364,B 18.9216,C -0.3983,E1 18.8762,E2 197.6717} C_DIS
LIN {X -37.0926,Y -125.3041,Z 156,A -107.2857,B 18.9216,C -0.3996,E1 18.8818,E2 195.5847} C_DIS
LIN {X -33.397,Y -126.339,Z 156,A -105.6379,B 18.9216,C -0.3972,E1 18.8862,E2 193.9409} C_DIS
LIN {X -29.5862,Y -127.2861,Z 156,A -103.6709,B 18.9214,C -0.4057,E1 18.8917,E2 191.9442} C_DIS
LIN {X -24.6448,Y -128.3336,Z 156,A -101.7077,B 18.9216,C -0.395,E1 18.897,E2 190.0108} C_DIS
LIN {X -22.0666,Y -128.8032,Z 156,A -99.9001,B 18.9211,C -0.4201,E1 18.9022,E2 188.1233} C_DIS
LIN {X -17.0886,Y -129.5564,Z 156,A -98.2495,B 18.9216,C -0.3979,E1 18.9065,E2 186.5395} C_DIS
LIN {X -12.7098,Y -130.0592,Z 156,A -96.3931,B 18.9216,C -0.3947,E1 18.9117,E2 184.6917} C_DIS
LIN {X -8.7967,Y -130.3842,Z 156,A -94.6081,B 18.9216,C -0.397,E1 18.9167,E2 182.8985} C_DIS
LIN {X -4.9387,Y -130.5854,Z 156,A -92.9201,B 18.9216,C -0.397,E1 18.9214,E2 181.2104} C_DIS
LIN {X -0.9263,Y -130.6756,Z 156,A -91.2156,B 18.9216,C -0.395,E1 18.9261,E2 179.5117} C_DIS
LIN {X -0.9263,Y -130.6756,Z 156,A -91.2156,B 18.9216,C -0.395,E1 18.9261,E2 179.5117} C_DIS
Enddeposition()
LIN {X 0.9038,Y -129.7407,Z 156,A -90.2126,B 16.1509,C -0.0837,E1 16.152,E2 179.3401} C_DIS
Startdeposition()
$VEL.CP = VEL_PRINT
LIN {X -2.8106,Y -129.7162,Z 156,A -92.0132,B 16.1509,C -0.0782,E1 16.1469,E2 181.1604} C_DIS
LIN {X -7.1476,Y -129.5494,Z 156,A -93.9336,B 16.1509,C -0.078,E1 16.1415,E2 183.0821} C_DIS
LIN {X -10.9861,Y -129.2789,Z 156,A -95.5369,B 16.1509,C -0.0813,E1 16.1371,E2 184.6748} C_DIS
LIN {X -16.4666,Y -128.6962,Z 156,A -98.6283,B 16.1509,C -0.0607,E1 16.1283,E2 187.8437} C_DIS
LIN {X -21.4477,Y -127.9598,Z 156,A -100.1694,B 16.1509,C -0.0832,E1 16.1243,E2 189.3058} C_DIS
LIN {X -25.0947,Y -127.2967,Z 156,A -101.8875,B 16.1509,C -0.0812,E1 16.1195,E2 191.0339} C_DIS
LIN {X -27.7483,Y -126.7432,Z 156,A -103.0317,B 16.1509,C -0.0835,E1 16.1164,E2 192.1721} C_DIS
LIN {X -31.9916,Y -125.7387,Z 156,A -104.9761,B 16.1509,C -0.084,E1 16.1111,E2 194.119} C_DIS
LIN {X -35.6064,Y -124.765,Z 156,A -106.6404,B 16.1509,C -0.0847,E1 16.1066,E2 195.7849} C_DIS
LIN {X -39.6326,Y -123.5432,Z 156,A -108.4526,B 16.1509,C -0.0876,E1 16.1018,E2 197.5918} C_DIS
LIN {X -42.712,Y -122.5127,Z 156,A -109.8866,B 16.1509,C -0.0888,E1 16.098,E2 199.0259} C_DIS
LIN {X -45.6996,Y -121.4299,Z 156,A -112.4324,B 16.151,C -0.0544,E1 16.0911,E2 201.7039} C_DIS
LIN {X -52.4891,Y -118.6541,Z 156,A -114.4431,B 16.1508,C -0.096,E1 16.0863,E2 203.5723} C_DIS
LIN {X -54.4266,Y -117.7767,Z 156,A -115.6116,B 16.1508,C -0.0899,E1 16.0832,E2 204.7675} C_DIS
LIN {X -57.5993,Y -116.2582,Z 156,A -117.0452,B 16.1508,C -0.0954,E1 16.0797,E2 206.1869} C_DIS
LIN {X -60.1541,Y -114.957,Z 156,A -118.2958,B 16.1508,C -0.0975,E1 16.0766,E2 207.4356} C_DIS
LIN {X -63.7612,Y -112.9986,Z 156,A -120.2615,B 16.1508,C -0.0952,E1 16.0717,E2 209.4188} C_DIS
LIN {X -70.5122,Y -108.9136,Z 156,A -123.531,B 16.1508,C -0.1068,E1 16.064,E2 212.6624} C_DIS
LIN {X -73.9202,Y -106.6301,Z 156,A -125.4438,B 16.1508,C -0.1066,E1 16.0595,E2 214.5864} C_DIS
LIN {X -77.0808,Y -104.3684,Z 156,A -127.2613,B 16.1508,C -0.1063,E1 16.0554,E2 216.4152} C_DIS
LIN {X -80.4389,Y -101.8029,Z 156,A -129.2052,B 16.1508,C -0.1072,E1 16.0511,E2 218.3673} C_DIS
LIN {X -83.8289,Y -99.0298,Z 156,A -131.1576,B 16.1508,C -0.1102,E1 16.0469,E2 220.321} C_DIS
LIN {X -87.1288,Y -96.1389,Z 156,A -133.0762,B 16.1507,C -0.1144,E1 16.0429,E2 222.2363} C_DIS
LIN {X -90.2623,Y -93.2032,Z 156,A -134.9555,B 16.1507,C -0.1187,E1 16.0391,E2 224.1127} C_DIS
LIN {X -93.4359,Y -90.0219,Z 156,A -136.9955,B 16.1507,C -0.1211,E1 16.0351,E2 226.158} C_DIS
LIN {X -96.6967,Y -86.5093,Z 156,A -139.1083,B 16.1507,C -0.1258,E1 16.0311,E2 228.269} C_DIS
LIN {X -99.6104,Y -83.1384,Z 156,A -141.3691,B 16.1507,C -0.1214,E1 16.027,E2 230.5623} C_DIS
LIN {X -101.8408,Y -80.3907,Z 156,A -142.5371,B 16.1505,C -0.1367,E1 16.0251,E2 231.6837} C_DIS
LIN {X -104.107,Y -77.4328,Z 156,A -144.2224,B 16.1505,C -0.1394,E1 16.0222,E2 233.3724} C_DIS
LIN {X -106.3081,Y -74.383,Z 156,A -146.1699,B 16.1505,C -0.1349,E1 16.019,E2 235.3517} C_DIS
LIN {X -108.3383,Y -71.3928,Z 156,A -147.5891,B 16.1505,C -0.144,E1 16.0169,E2 236.7492} C_DIS
LIN {X -110.6831,Y -67.7009,Z 156,A -149.5708,B 16.1505,C -0.1473,E1 16.0139,E2 238.735} C_DIS
LIN {X -113.1453,Y -63.5001,Z 156,A -151.725,B 16.1504,C -0.1527,E1 16.0109,E2 240.8879} C_DIS
LIN {X -115.1058,Y -59.8707,Z 156,A -153.5403,B 16.1504,C -0.1577,E1 16.0085,E2 242.7007} C_DIS
LIN {X -117.3983,Y -55.2428,Z 156,A -155.7543,B 16.1503,C -0.1657,E1 16.0059,E2 244.9048} C_DIS
LIN {X -118.8242,Y -52.1045,Z 156,A -157.2989,B 16.1503,C -0.1692,E1 16.0041,E2 246.4506} C_DIS
LIN {X -120.2796,Y -48.6463,Z 156,A -158.9929,B 16.1502,C -0.1727,E1 16.0023,E2 248.1471} C_DIS
LIN {X -121.5314,Y -45.4286,Z 156,A -160.8192,B 16.1502,C -0.1682,E1 16.0004,E2 250.0064} C_DIS
LIN {X -122.6217,Y -42.3976,Z 156,A -161.902,B 16.1501,C -0.1821,E1 15.9995,E2 251.0487} C_DIS
LIN {X -123.6299,Y -39.3613,Z 156,A -163.3881,B 16.1501,C -0.1839,E1 15.9982,E2 252.5417} C_DIS
LIN {X -124.6768,Y -35.9121,Z 156,A -164.9653,B 16.1501,C -0.1889,E1 15.9969,E2 254.1156} C_DIS
LIN {X -125.6382,Y -32.3872,Z 156,A -166.711,B 16.1501,C -0.1898,E1 15.9957,E2 255.8746} C_DIS
LIN {X -126.6008,Y -28.3931,Z 156,A -168.5218,B 16.1499,C -0.1952,E1 15.9945,E2 257.6829} C_DIS
LIN {X -127.2703,Y -25.2266,Z 156,A -169.84,B 16.1499,C -0.2026,E1 15.9938,E2 258.9868} C_DIS
LIN {X -127.8568,Y -22.0648,Z 156,A -171.2924,B 16.1499,C -0.2059,E1 15.9931,E2 260.4412} C_DIS
LIN {X -128.3447,Y -19.0204,Z 156,A -172.8919,B 16.1499,C -0.2031,E1 15.9924,E2 262.0663} C_DIS
LIN {X -128.9789,Y -14.0785,Z 156,A -174.6569,B 16.1496,C -0.2223,E1 15.9918,E2 263.7786} C_DIS
LIN {X -129.2451,Y -11.3861,Z 156,A -176.2245,B 16.1496,C -0.2151,E1 15.9914,E2 265.3876} C_DIS
LIN {X -129.504,Y -7.9026,Z 156,A -177.6888,B 16.1496,C -0.222,E1 15.9911,E2 266.841} C_DIS
LIN {X -129.7044,Y -3.2602,Z 156,A -179.6241,B 16.1495,C -0.2316,E1 15.9909,E2 268.7603} C_DIS
LIN {X -129.7436,Y -0.6031,Z 156,A 179.0628,B 16.1495,C -0.2311,E1 15.9909,E2 270.0878} C_DIS
LIN {X -129.674,Y 4.3388,Z 156,A 176.9364,B 16.1494,C -0.2394,E1 15.991,E2 272.205} C_DIS
LIN {X -129.3523,Y 10.1072,Z 156,A 174.1724,B 16.1494,C -0.241,E1 15.9915,E2 274.99} C_DIS
LIN {X -128.9739,Y 14.1253,Z 156,A 172.453,B 16.1492,C -0.2482,E1 15.992,E2 276.6998} C_DIS
LIN {X -128.5356,Y 17.6851,Z 156,A 170.9494,B 16.1492,C -0.2553,E1 15.9925,E2 278.1922} C_DIS
LIN {X -128.0483,Y 20.917,Z 156,A 169.4619,B 16.1491,C -0.2584,E1 15.9931,E2 279.6828} C_DIS
LIN {X -127.5026,Y 24.0187,Z 156,A 168.2176,B 16.1489,C -0.2669,E1 15.9938,E2 280.9084} C_DIS
LIN {X -127.055,Y 26.2849,Z 156,A 166.9227,B 16.149,C -0.262,E1 15.9945,E2 282.2334} C_DIS
LIN {X -126.1697,Y 30.2471,Z 156,A 165.0857,B 16.149,C -0.2661,E1 15.9956,E2 284.0728} C_DIS
LIN {X -125.2784,Y 33.7506,Z 156,A 163.624,B 16.1488,C -0.2747,E1 15.9967,E2 285.517} C_DIS
LIN {X -124.5268,Y 36.4243,Z 156,A 162.3519,B 16.1488,C -0.277,E1 15.9976,E2 286.7926} C_DIS
LIN {X -123.3785,Y 40.1482,Z 156,A 160.447,B 16.1488,C -0.2767,E1 15.9993,E2 288.7162} C_DIS
LIN {X -122.1113,Y 43.8461,Z 156,A 158.8122,B 16.1487,C -0.2844,E1 16.0008,E2 290.3381} C_DIS
LIN {X -120.6584,Y 47.7046,Z 156,A 157.0332,B 16.1485,C -0.2908,E1 16.0025,E2 292.1099} C_DIS
LIN {X -119.7122,Y 50.0261,Z 156,A 155.8657,B 16.1485,C -0.2923,E1 16.0038,E2 293.2827} C_DIS
LIN {X -118.1014,Y 53.7245,Z 156,A 153.5767,B 16.1487,C -0.2827,E1 16.0065,E2 295.6269} C_DIS
LIN {X -116.3303,Y 57.4532,Z 156,A 152.241,B 16.1483,C -0.3018,E1 16.0081,E2 296.9049} C_DIS
LIN {X -113.8002,Y 62.3192,Z 156,A 149.8799,B 16.1482,C -0.3102,E1 16.0111,E2 299.2558} C_DIS
LIN {X -112.6522,Y 64.3708,Z 156,A 148.3906,B 16.1484,C -0.2999,E1 16.0133,E2 300.7949} C_DIS
LIN {X -110.8207,Y 67.4762,Z 156,A 147.0274,B 16.1482,C -0.3108,E1 16.0152,E2 302.13} C_DIS
LIN {X -108.6475,Y 70.922,Z 156,A 145.2449,B 16.1481,C -0.3159,E1 16.0179,E2 303.9083} C_DIS
LIN {X -106.5549,Y 74.0282,Z 156,A 143.598,B 16.148,C -0.3204,E1 16.0205,E2 305.5522} C_DIS
LIN {X -103.9351,Y 77.6637,Z 156,A 141.5745,B 16.148,C -0.3241,E1 16.0238,E2 307.5781} C_DIS
LIN {X -101.238,Y 81.1489,Z 156,A 139.672,B 16.1478,C -0.3302,E1 16.0271,E2 309.4731} C_DIS
LIN {X -98.7354,Y 84.1752,Z 156,A 137.8967,B 16.1478,C -0.3331,E1 16.0303,E2 311.2509} C_DIS
LIN {X -95.9734,Y 87.3112,Z 156,A 136.0424,B 16.1477,C -0.3372,E1 16.0337,E2 313.1038} C_DIS
LIN {X -92.9459,Y 90.528,Z 156,A 134.0559,B 16.1476,C -0.3406,E1 16.0375,E2 315.0919} C_DIS
LIN {X -90.035,Y 93.4232,Z 156,A 132.2204,B 16.1476,C -0.3439,E1 16.0412,E2 316.9277} C_DIS
LIN {X -86.8318,Y 96.4079,Z 156,A 130.2465,B 16.1475,C -0.3468,E1 16.0453,E2 318.9038} C_DIS
LIN {X -83.599,Y 99.224,Z 156,A 128.404,B 16.1474,C -0.3522,E1 16.0492,E2 320.7383} C_DIS
LIN {X -80.3716,Y 101.8558,Z 156,A 126.5156,B 16.1474,C -0.3544,E1 16.0533,E2 322.6301} C_DIS
LIN {X -76.8952,Y 104.5048,Z 156,A 124.6766,B 16.1472,C -0.3608,E1 16.0574,E2 324.4566} C_DIS
LIN {X -73.7561,Y 106.7442,Z 156,A 122.8244,B 16.1472,C -0.3595,E1 16.0616,E2 326.3238} C_DIS
LIN {X -70.1097,Y 109.1732,Z 156,A 120.9145,B 16.1472,C -0.3636,E1 16.0661,E2 328.2287} C_DIS
LIN {X -66.3111,Y 111.5212,Z 156,A 118.9359,B 16.147,C -0.3667,E1 16.0708,E2 330.2059} C_DIS
LIN {X -62.1837,Y 113.8741,Z 156,A 116.8103,B 16.147,C -0.3692,E1 16.076,E2 332.3324} C_DIS
LIN {X -58.7762,Y 115.6675,Z 156,A 115.2112,B 16.1469,C -0.3748,E1 16.0799,E2 333.9182} C_DIS
LIN {X -55.4958,Y 117.2777,Z 156,A 113.587,B 16.1469,C -0.3768,E1 16.084,E2 335.542} C_DIS
LIN {X -52.178,Y 118.7924,Z 156,A 111.6872,B 16.1469,C -0.3702,E1 16.0889,E2 337.4731} C_DIS
LIN {X -47.9919,Y 120.5434,Z 156,A 109.9797,B 16.1467,C -0.3817,E1 16.0933,E2 339.1451} C_DIS
LIN {X -45.1736,Y 121.6269,Z 156,A 108.6102,B 16.1467,C -0.3822,E1 16.0968,E2 340.5176} C_DIS
LIN {X -40.8513,Y 123.1456,Z 156,A 106.5781,B 16.1467,C -0.3841,E1 16.1022,E2 342.5489} C_DIS
LIN {X -37.6905,Y 124.1497,Z 156,A 105.1078,B 16.1467,C -0.3854,E1 16.1061,E2 344.0186} C_DIS
LIN {X -34.0143,Y 125.208,Z 156,A 103.3339,B 16.1467,C -0.3843,E1 16.1109,E2 345.8009} C_DIS
LIN {X -29.6234,Y 126.3197,Z 156,A 101.3541,B 16.1466,C -0.3866,E1 16.1163,E2 347.7767} C_DIS
LIN {X -22.4371,Y 127.7906,Z 156,A 98.2488,B 16.1464,C -0.393,E1 16.1247,E2 350.8645} C_DIS
LIN {X -19.6607,Y 128.2466,Z 156,A 96.9111,B 16.1464,C -0.3908,E1 16.1284,E2 352.2122} C_DIS
LIN {X -14.0591,Y 128.981,Z 156,A 93.9855,B 16.1468,C -0.3785,E1 16.1367,E2 355.1851} C_DIS
LIN {X -10.0341,Y 129.3576,Z 156,A 92.5715,B 16.1465,C -0.3907,E1 16.1405,E2 356.5561} C_DIS
LIN {X -6.3709,Y 129.5885,Z 156,A 90.9836,B 16.1465,C -0.3922,E1 16.1449,E2 358.1392} C_DIS
LIN {X -2.5084,Y 129.7212,Z 156,A 89.2022,B 16.1465,C -0.3902,E1 16.1499,E2 359.9283} C_DIS
LIN {X 1.238,Y 129.7401,Z 156,A 87.1758,B 16.1468,C -0.3785,E1 16.1557,E2 361.9961} C_DIS
LIN {X 5.3372,Y 129.6354,Z 156,A 85.9111,B 16.1464,C -0.3959,E1 16.1591,E2 363.198} C_DIS
LIN {X 8.7533,Y 129.4511,Z 156,A 83.764,B 16.1468,C -0.3755,E1 16.1652,E2 365.4169} C_DIS
LIN {X 13.3096,Y 129.0616,Z 156,A 82.4305,B 16.1463,C -0.397,E1 16.1687,E2 366.6717} C_DIS
LIN {X 18.6186,Y 128.4022,Z 156,A 80.0015,B 16.1464,C -0.3942,E1 16.1755,E2 369.1076} C_DIS
LIN {X 23.905,Y 127.5243,Z 156,A 77.7359,B 16.1464,C -0.3965,E1 16.1817,E2 371.3611} C_DIS
LIN {X 27.1674,Y 126.8687,Z 156,A 76.0448,B 16.1465,C -0.3885,E1 16.1864,E2 373.0772} C_DIS
LIN {X 30.719,Y 126.056,Z 156,A 74.5204,B 16.1465,C -0.3903,E1 16.1905,E2 374.5917} C_DIS
LIN {X 33.7255,Y 125.2851,Z 156,A 73.0325,B 16.1466,C -0.3856,E1 16.1945,E2 376.0928} C_DIS
LIN {X 37.9668,Y 124.0652,Z 156,A 71.197,B 16.1466,C -0.3878,E1 16.1994,E2 377.9151} C_DIS
LIN {X 41.204,Y 123.0281,Z 156,A 69.6943,B 16.1466,C -0.3865,E1 16.2034,E2 379.4179} C_DIS
LIN {X 48.8015,Y 120.2171,Z 156,A 66.1579,B 16.1466,C -0.3843,E1 16.2126,E2 382.9497} C_DIS
LIN {X 52.1508,Y 118.8041,Z 156,A 64.36,B 16.1468,C -0.3762,E1 16.2173,E2 384.7699} C_DIS
LIN {X 56.2682,Y 116.9087,Z 156,A 62.5662,B 16.1468,C -0.3807,E1 16.2218,E2 386.5401} C_DIS
LIN {X 59.757,Y 115.1656,Z 156,A 60.8612,B 16.1468,C -0.3791,E1 16.226,E2 388.2433} C_DIS
LIN {X 62.6186,Y 113.6358,Z 156,A 58.7697,B 16.1473,C -0.3552,E1 16.2313,E2 390.4105} C_DIS
LIN {X 66.9127,Y 111.1613,Z 156,A 57.3352,B 16.1468,C -0.3771,E1 16.2346,E2 391.7593} C_DIS
LIN {X 69.2085,Y 109.7465,Z 156,A 55.9172,B 16.147,C -0.3677,E1 16.238,E2 393.2038} C_DIS
LIN {X 73.1357,Y 107.17,Z 156,A 53.8905,B 16.147,C -0.366,E1 16.2427,E2 395.2257} C_DIS
LIN {X 76.6613,Y 104.6766,Z 156,A 52.0619,B 16.147,C -0.3654,E1 16.2468,E2 397.0459} C_DIS
LIN {X 79.8644,Y 102.2542,Z 156,A 50.2438,B 16.1472,C -0.3608,E1 16.2508,E2 398.8699} C_DIS
LIN {X 82.8004,Y 99.891,Z 156,A 48.6098,B 16.1472,C -0.3588,E1 16.2544,E2 400.5012} C_DIS
LIN {X 86.0032,Y 97.1471,Z 156,A 46.7455,B 16.1472,C -0.3551,E1 16.2583,E2 402.3666} C_DIS
LIN {X 89.4357,Y 93.9971,Z 156,A 44.9314,B 16.1472,C -0.3594,E1 16.2619,E2 404.1536} C_DIS
LIN {X 91.6635,Y 91.826,Z 156,A 43.315,B 16.1474,C -0.3482,E1 16.2652,E2 405.7988} C_DIS
LIN {X 94.7437,Y 88.6444,Z 156,A 41.3533,B 16.1475,C -0.3439,E1 16.269,E2 407.7625} C_DIS
LIN {X 97.7297,Y 85.3406,Z 156,A 39.4397,B 16.1475,C -0.3414,E1 16.2725,E2 409.6712} C_DIS
LIN {X 100.5021,Y 82.0576,Z 156,A 37.6195,B 16.1476,C -0.3397,E1 16.2758,E2 411.4837} C_DIS
LIN {X 102.9691,Y 78.9398,Z 156,A 35.7874,B 16.1477,C -0.333,E1 16.2789,E2 413.326} C_DIS
LIN {X 108.1645,Y 71.6559,Z 156,A 31.8656,B 16.1479,C -0.3244,E1 16.2852,E2 417.2475} C_DIS
LIN {X 110.5316,Y 67.9477,Z 156,A 30.0634,B 16.1479,C -0.3244,E1 16.2879,E2 419.0351} C_DIS
LIN {X 112.4989,Y 64.6395,Z 156,A 28.2823,B 16.1481,C -0.3172,E1 16.2904,E2 420.8271} C_DIS
LIN {X 114.4326,Y 61.1504,Z 156,A 25.5594,B 16.1487,C -0.2793,E1 16.2942,E2 423.6622} C_DIS
LIN {X 117.56,Y 54.8953,Z 156,A 23.5478,B 16.1482,C -0.3084,E1 16.2964,E2 425.5528} C_DIS
LIN {X 118.5972,Y 52.6162,Z 156,A 22.3306,B 16.1484,C -0.3015,E1 16.2978,E2 426.784} C_DIS
LIN {X 119.9442,Y 49.4706,Z 156,A 20.9659,B 16.1484,C -0.3024,E1 16.2993,E2 428.1333} C_DIS
LIN {X 120.9935,Y 46.8426,Z 156,A 19.7304,B 16.1484,C -0.2995,E1 16.3005,E2 429.3684} C_DIS
LIN {X 122.0458,Y 44.0278,Z 156,A 18.3893,B 16.1484,C -0.2952,E1 16.3018,E2 430.7125} C_DIS
LIN {X 123.2919,Y 40.4119,Z 156,A 16.5509,B 16.1486,C -0.2851,E1 16.3035,E2 432.5702} C_DIS
LIN {X 124.5426,Y 36.3703,Z 156,A 14.8424,B 16.1486,C -0.2854,E1 16.3048,E2 434.2621} C_DIS
LIN {X 125.5749,Y 32.6362,Z 156,A 12.9544,B 16.1488,C -0.2742,E1 16.3062,E2 436.1727} C_DIS
LIN {X 126.8998,Y 27.023,Z 156,A 10.2007,B 16.1491,C -0.2594,E1 16.3079,E2 438.9533} C_DIS
LIN {X 127.6734,Y 23.0922,Z 156,A 9.1421,B 16.1487,C -0.2793,E1 16.3084,E2 439.9311} C_DIS
LIN {X 128.861,Y 15.1202,Z 156,A 4.6662,B 16.1494,C -0.2362,E1 16.3102,E2 444.5181} C_DIS
LIN {X 129.3748,Y 9.7991,Z 156,A 3.2336,B 16.149,C -0.2619,E1 16.3105,E2 445.8456} C_DIS
LIN {X 129.6042,Y 6.0589,Z 156,A 1.4346,B 16.1492,C -0.2517,E1 16.3108,E2 447.6637} C_DIS
LIN {X 129.7232,Y 2.3862,Z 156,A -0.2365,B 16.1492,C -0.2451,E1 16.3108,E2 449.3425} C_DIS
LIN {X 129.7346,Y -1.7013,Z 156,A -2.0362,B 16.1494,C -0.2398,E1 16.3108,E2 451.1439} C_DIS
LIN {X 129.638,Y -5.2695,Z 156,A -3.6314,B 16.1494,C -0.2343,E1 16.3108,E2 452.7434} C_DIS
LIN {X 129.2478,Y -11.3543,Z 156,A -7.059,B 16.1499,C -0.2001,E1 16.3099,E2 456.2601} C_DIS
LIN {X 128.5886,Y -17.2879,Z 156,A -8.7874,B 16.1496,C -0.2242,E1 16.3094,E2 457.8863} C_DIS
LIN {X 127.8013,Y -22.3777,Z 156,A -10.9427,B 16.1496,C -0.2216,E1 16.3084,E2 460.0307} C_DIS
LIN {X 127.323,Y -24.9579,Z 156,A -12.4713,B 16.1498,C -0.2049,E1 16.3076,E2 461.6043} C_DIS
LIN {X 126.5914,Y -28.4343,Z 156,A -13.8208,B 16.1498,C -0.208,E1 16.3068,E2 462.9302} C_DIS
LIN {X 125.6832,Y -32.21,Z 156,A -15.5155,B 16.1498,C -0.2036,E1 16.3057,E2 464.625} C_DIS
LIN {X 124.3587,Y -36.9985,Z 156,A -17.6506,B 16.1498,C -0.1992,E1 16.304,E2 466.7562} C_DIS
LIN {X 123.1962,Y -40.6993,Z 156,A -19.3494,B 16.1499,C -0.1946,E1 16.3026,E2 468.4556} C_DIS
LIN {X 121.9691,Y -44.2407,Z 156,A -21.7785,B 16.1503,C -0.1625,E1 16.3002,E2 470.9775} C_DIS
LIN {X 119.9012,Y -49.5735,Z 156,A -23.3465,B 16.15,C -0.189,E1 16.2987,E2 472.4369} C_DIS
LIN {X 118.1677,Y -53.5766,Z 156,A -25.4855,B 16.1502,C -0.176,E1 16.2962,E2 474.6037} C_DIS
LIN {X 115.9216,Y -58.2771,Z 156,A -27.6115,B 16.1502,C -0.1757,E1 16.2937,E2 476.7123} C_DIS
LIN {X 114.4667,Y -61.0871,Z 156,A -29.13,B 16.1502,C -0.1675,E1 16.2917,E2 478.247} C_DIS
LIN {X 112.4818,Y -64.6693,Z 156,A -31.0008,B 16.1503,C -0.1604,E1 16.2891,E2 480.1277} C_DIS
LIN {X 110.0476,Y -68.7291,Z 156,A -33.0437,B 16.1503,C -0.1565,E1 16.2861,E2 482.1679} C_DIS
LIN {X 107.6741,Y -72.3918,Z 156,A -34.9811,B 16.1504,C -0.1511,E1 16.2831,E2 484.1091} C_DIS
LIN {X 104.2664,Y -77.2189,Z 156,A -37.4584,B 16.1504,C -0.149,E1 16.2791,E2 486.5743} C_DIS
LIN {X 102.1156,Y -80.0408,Z 156,A -39.0451,B 16.1504,C -0.1444,E1 16.2764,E2 488.1654} C_DIS
LIN {X 99.5611,Y -83.1971,Z 156,A -40.9285,B 16.1505,C -0.1369,E1 16.273,E2 490.0618} C_DIS
LIN {X 95.7739,Y -87.5306,Z 156,A -43.4038,B 16.1505,C -0.1331,E1 16.2684,E2 492.5325} C_DIS
LIN {X 92.8376,Y -90.6387,Z 156,A -45.2307,B 16.1505,C -0.1309,E1 16.2649,E2 494.3546} C_DIS
LIN {X 89.4231,Y -94.0089,Z 156,A -47.3806,B 16.1506,C -0.1251,E1 16.2606,E2 496.5109} C_DIS
LIN {X 86.1948,Y -96.9778,Z 156,A -49.3084,B 16.1506,C -0.1212,E1 16.2566,E2 498.44} C_DIS
LIN {X 82.9631,Y -99.7562,Z 156,A -51.1593,B 16.1506,C -0.1184,E1 16.2527,E2 500.2895} C_DIS
LIN {X 78.8681,Y -103.024,Z 156,A -53.4547,B 16.1506,C -0.1144,E1 16.2476,E2 502.5855} C_DIS
LIN {X 75.3629,Y -105.6152,Z 156,A -55.2732,B 16.1506,C -0.1144,E1 16.2435,E2 504.3937} C_DIS
LIN {X 72.2451,Y -107.7721,Z 156,A -56.9221,B 16.1507,C -0.1122,E1 16.2397,E2 506.0415} C_DIS
LIN {X 69.0938,Y -109.8189,Z 156,A -58.6105,B 16.1507,C -0.1082,E1 16.2358,E2 507.7352} C_DIS
LIN {X 66.7651,Y -111.2506,Z 156,A -59.8897,B 16.1507,C -0.1037,E1 16.2327,E2 509.0242} C_DIS
LIN {X 63.042,Y -113.4014,Z 156,A -62.1145,B 16.1509,C -0.0894,E1 16.2272,E2 511.2893} C_DIS
LIN {X 59.6,Y -115.2475,Z 156,A -64.2091,B 16.1509,C -0.0743,E1 16.2218,E2 513.4288} C_DIS
LIN {X 54.4446,Y -117.7684,Z 156,A -65.697,B 16.1508,C -0.1061,E1 16.2184,E2 514.7965} C_DIS
LIN {X 49.7456,Y -119.8293,Z 156,A -68.1169,B 16.1508,C -0.0977,E1 16.2122,E2 517.2368} C_DIS
LIN {X 46.9128,Y -120.9662,Z 156,A -69.5586,B 16.1508,C -0.0929,E1 16.2084,E2 518.6908} C_DIS
LIN {X 43.5147,Y -122.2308,Z 156,A -71.1047,B 16.1508,C -0.0929,E1 16.2043,E2 520.2319} C_DIS
LIN {X 36.8621,Y -124.3986,Z 156,A -74.0229,B 16.1508,C -0.0952,E1 16.1966,E2 523.1326} C_DIS
LIN {X 32.8661,Y -125.5142,Z 156,A -76.1331,B 16.1508,C -0.0841,E1 16.1908,E2 525.2771} C_DIS
LIN {X 25.1767,Y -127.2805,Z 156,A -79.4481,B 16.1508,C -0.0869,E1 16.1819,E2 528.5749} C_DIS
LIN {X 17.6034,Y -128.5472,Z 156,A -82.8384,B 16.1508,C -0.0847,E1 16.1725,E2 531.9677} C_DIS
LIN {X 14.6537,Y -128.9166,Z 156,A -84.3361,B 16.1509,C -0.0779,E1 16.1683,E2 533.488} C_DIS
LIN {X 10.6831,Y -129.3045,Z 156,A -85.9362,B 16.1509,C -0.0825,E1 16.1639,E2 535.0701} C_DIS
LIN {X 6.7756,Y -129.5681,Z 156,A -87.6611,B 16.1509,C -0.082,E1 16.1591,E2 536.7955} C_DIS
LIN {X 3.4036,Y -129.7005,Z 156,A -89.2364,B 16.1509,C -0.0788,E1 16.1546,E2 538.3815} C_DIS
LIN {X 3.4036,Y -129.7005,Z 156,A -89.2364,B 16.1509,C -0.0788,E1 16.1546,E2 538.3815} C_DIS
Enddeposition()
LIN {X 0.8932,Y -128.8057,Z 156,A -89.7423,B 16.1507,C -0.1086,E1 16.1535,E2 538.7802} C_DIS
Startdeposition()
$VEL.CP = VEL_PRINT
LIN {X 4.7576,Y -128.7235,Z 156,A -87.9303,B 16.1507,C -0.1121,E1 16.1586,E2 536.9565} C_DIS
LIN {X 7.8986,Y -128.5687,Z 156,A -86.4766,B 16.1507,C -0.1144,E1 16.1627,E2 535.4955} C_DIS
LIN {X 12.1743,Y -128.2345,Z 156,A -84.8763,B 16.1507,C -0.105,E1 16.1671,E2 533.9303} C_DIS
LIN {X 15.3142,Y -127.8975,Z 156,A -83.1518,B 16.1507,C -0.1163,E1 16.1719,E2 532.1672} C_DIS
LIN {X 18.9568,Y -127.4106,Z 156,A -81.5948,B 16.1507,C -0.1146,E1 16.1762,E2 530.6184} C_DIS
LIN {X 22.4786,Y -126.8346,Z 156,A -79.9418,B 16.1507,C -0.1179,E1 16.1808,E2 528.9565} C_DIS
LIN {X 26.6563,Y -126.0237,Z 156,A -78.1237,B 16.1507,C -0.1168,E1 16.1858,E2 527.1459} C_DIS
LIN {X 30.1302,Y -125.2374,Z 156,A -76.441,B 16.1507,C -0.1215,E1 16.1904,E2 525.4502} C_DIS
LIN {X 34.345,Y -124.1482,Z 156,A -74.6138,B 16.1507,C -0.1196,E1 16.1953,E2 523.6344} C_DIS
LIN {X 37.7922,Y -123.1421,Z 156,A -73.023,B 16.1507,C -0.1211,E1 16.1995,E2 522.043} C_DIS
LIN {X 40.7898,Y -122.1819,Z 156,A -71.6195,B 16.1507,C -0.1227,E1 16.2033,E2 520.6379} C_DIS
LIN {X 44.4564,Y -120.8984,Z 156,A -69.7693,B 16.1506,C -0.1289,E1 16.2082,E2 518.7717} C_DIS
LIN {X 47.8244,Y -119.6041,Z 156,A -68.3095,B 16.1506,C -0.126,E1 16.2119,E2 517.3275} C_DIS
LIN {X 50.7633,Y -118.3868,Z 156,A -66.9036,B 16.1506,C -0.1276,E1 16.2155,E2 515.9214} C_DIS
LIN {X 53.6379,Y -117.1127,Z 156,A -65.5132,B 16.1506,C -0.1292,E1 16.2191,E2 514.5306} C_DIS
LIN {X 56.4783,Y -115.77,Z 156,A -64.1259,B 16.1506,C -0.1309,E1 16.2226,E2 513.1431} C_DIS
LIN {X 59.6661,Y -114.1586,Z 156,A -62.5991,B 16.1506,C -0.1313,E1 16.2263,E2 511.622} C_DIS
LIN {X 62.3901,Y -112.695,Z 156,A -61.1406,B 16.1506,C -0.1363,E1 16.2299,E2 510.1523} C_DIS
LIN {X 65.2477,Y -111.0649,Z 156,A -59.8164,B 16.1506,C -0.1339,E1 16.2331,E2 508.8429} C_DIS
LIN {X 67.5985,Y -109.6504,Z 156,A -58.4954,B 16.1506,C -0.1395,E1 16.2363,E2 507.5088} C_DIS
LIN {X 70.248,Y -107.9718,Z 156,A -57.108,B 16.1505,C -0.1417,E1 16.2396,E2 506.1206} C_DIS
LIN {X 73.2414,Y -105.9648,Z 156,A -55.5115,B 16.1505,C -0.1444,E1 16.2432,E2 504.5231} C_DIS
LIN {X 76.3648,Y -103.7358,Z 156,A -53.7402,B 16.1505,C -0.15,E1 16.2473,E2 502.7422} C_DIS
LIN {X 79.8588,Y -101.0712,Z 156,A -51.7491,B 16.1504,C -0.1551,E1 16.2517,E2 500.7445} C_DIS
LIN {X 82.9316,Y -98.565,Z 156,A -50.0887,B 16.1504,C -0.1551,E1 16.2552,E2 499.0942} C_DIS
LIN {X 85.9088,Y -95.981,Z 156,A -48.3407,B 16.1504,C -0.1587,E1 16.2589,E2 497.3447} C_DIS
LIN {X 88.8038,Y -93.3093,Z 156,A -46.5864,B 16.1504,C -0.1626,E1 16.2625,E2 495.588} C_DIS
LIN {X 91.6405,Y -90.5253,Z 156,A -44.7647,B 16.1502,C -0.1685,E1 16.2661,E2 493.7577} C_DIS
LIN {X 94.3661,Y -87.6798,Z 156,A -43.1115,B 16.1502,C -0.1691,E1 16.2692,E2 492.1141} C_DIS
LIN {X 97.0022,Y -84.7541,Z 156,A -41.2981,B 16.1502,C -0.1754,E1 16.2726,E2 490.2911} C_DIS
LIN {X 99.7152,Y -81.5449,Z 156,A -39.4585,B 16.1502,C -0.1789,E1 16.2759,E2 488.4525} C_DIS
LIN {X 102.5071,Y -78.0069,Z 156,A -37.4724,B 16.1501,C -0.1833,E1 16.2793,E2 486.466} C_DIS
LIN {X 105.039,Y -74.5631,Z 156,A -35.5714,B 16.1501,C -0.1881,E1 16.2824,E2 484.5624} C_DIS
LIN {X 107.3517,Y -71.193,Z 156,A -33.8713,B 16.1501,C -0.1887,E1 16.285,E2 482.8739} C_DIS
LIN {X 109.0631,Y -68.5418,Z 156,A -32.4242,B 16.15,C -0.194,E1 16.2872,E2 481.4197} C_DIS
LIN {X 111.2923,Y -64.8603,Z 156,A -30.5888,B 16.15,C -0.1963,E1 16.2898,E2 479.591} C_DIS
LIN {X 112.8494,Y -62.1112,Z 156,A -29.1906,B 16.1499,C -0.1999,E1 16.2917,E2 478.1918} C_DIS
LIN {X 114.5437,Y -58.9256,Z 156,A -27.5651,B 16.1499,C -0.2051,E1 16.2939,E2 476.5616} C_DIS
LIN {X 115.9635,Y -56.0805,Z 156,A -26.2112,B 16.1499,C -0.2069,E1 16.2955,E2 475.2129} C_DIS
LIN {X 117.2578,Y -53.3238,Z 156,A -24.8304,B 16.1497,C -0.2116,E1 16.2971,E2 473.8272} C_DIS
LIN {X 118.693,Y -50.0436,Z 156,A -23.4208,B 16.1497,C -0.2097,E1 16.2987,E2 472.4369} C_DIS
LIN {X 119.7562,Y -47.447,Z 156,A -22.0426,B 16.1497,C -0.2179,E1 16.3001,E2 471.0417} C_DIS
LIN {X 120.876,Y -44.5162,Z 156,A -20.4751,B 16.1495,C -0.2281,E1 16.3017,E2 469.4519} C_DIS
LIN {X 122.3098,Y -40.4057,Z 156,A -18.7449,B 16.1495,C -0.2264,E1 16.3032,E2 467.7434} C_DIS
LIN {X 123.2633,Y -37.3961,Z 156,A -17.3075,B 16.1495,C -0.2317,E1 16.3044,E2 466.3002} C_DIS
LIN {X 124.2684,Y -33.914,Z 156,A -15.7529,B 16.1495,C -0.2345,E1 16.3056,E2 464.7502} C_DIS
LIN {X 125.2202,Y -30.2017,Z 156,A -14.3009,B 16.1495,C -0.2306,E1 16.3066,E2 463.3255} C_DIS
LIN {X 125.7777,Y -27.796,Z 156,A -13.0438,B 16.1494,C -0.2395,E1 16.3073,E2 462.0483} C_DIS
LIN {X 126.4238,Y -24.6889,Z 156,A -11.6917,B 16.1494,C -0.2416,E1 16.3081,E2 460.7013} C_DIS
LIN {X 126.9886,Y -21.5942,Z 156,A -10.1919,B 16.1492,C -0.2494,E1 16.3088,E2 459.1877} C_DIS
LIN {X 127.4831,Y -18.4499,Z 156,A -8.9396,B 16.1492,C -0.2479,E1 16.3093,E2 457.9527} C_DIS
LIN {X 127.894,Y -15.3435,Z 156,A -7.3232,B 16.1491,C -0.2601,E1 16.3099,E2 456.3082} C_DIS
LIN {X 128.3316,Y -11.1077,Z 156,A -5.537,B 16.1491,C -0.262,E1 16.3104,E2 454.5322} C_DIS
LIN {X 128.5865,Y -7.6107,Z 156,A -3.8432,B 16.1489,C -0.2715,E1 16.3107,E2 452.8205} C_DIS
LIN {X 128.7446,Y -4.1867,Z 156,A -2.4953,B 16.1489,C -0.2699,E1 16.3108,E2 451.4915} C_DIS
LIN {X 128.8028,Y -1.574,Z 156,A -1.2896,B 16.1489,C -0.2749,E1 16.3108,E2 450.2792} C_DIS
LIN {X 128.7937,Y 2.1226,Z 156,A 0.3674,B 16.1487,C -0.2804,E1 16.3108,E2 448.6185} C_DIS
LIN {X 128.6562,Y 6.3186,Z 156,A 2.1884,B 16.1487,C -0.2844,E1 16.3106,E2 446.8007} C_DIS
LIN {X 128.405,Y 10.2382,Z 156,A 4.0685,B 16.1485,C -0.2945,E1 16.3103,E2 444.9027} C_DIS
LIN {X 128.0214,Y 14.2493,Z 156,A 5.738,B 16.1485,C -0.2955,E1 16.3098,E2 443.2454} C_DIS
LIN {X 127.6369,Y 17.364,Z 156,A 7.0206,B 16.1485,C -0.2956,E1 16.3093,E2 441.9745} C_DIS
LIN {X 127.1149,Y 20.8373,Z 156,A 8.604,B 16.1484,C -0.301,E1 16.3086,E2 440.3867} C_DIS
LIN {X 126.6385,Y 23.5658,Z 156,A 9.9251,B 16.1482,C -0.3079,E1 16.308,E2 439.0538} C_DIS
LIN {X 126.0258,Y 26.6468,Z 156,A 11.1884,B 16.1482,C -0.3072,E1 16.3073,E2 437.8045} C_DIS
LIN {X 125.2364,Y 30.1346,Z 156,A 12.8005,B 16.1482,C -0.3127,E1 16.3062,E2 436.188} C_DIS
LIN {X 124.266,Y 33.9231,Z 156,A 14.6193,B 16.148,C -0.3205,E1 16.3049,E2 434.3581} C_DIS
LIN {X 123.2664,Y 37.3861,Z 156,A 16.1723,B 16.148,C -0.3234,E1 16.3037,E2 432.809} C_DIS
LIN {X 122.1668,Y 40.835,Z 156,A 17.6702,B 16.148,C -0.324,E1 16.3024,E2 431.3226} C_DIS
LIN {X 120.8964,Y 44.4618,Z 156,A 19.4988,B 16.1478,C -0.333,E1 16.3006,E2 429.4784} C_DIS
LIN {X 119.6026,Y 47.8282,Z 156,A 20.9519,B 16.1478,C -0.3322,E1 16.2992,E2 428.0412} C_DIS
LIN {X 118.3643,Y 50.8152,Z 156,A 22.3876,B 16.1477,C -0.336,E1 16.2976,E2 426.6043} C_DIS
LIN {X 117.1216,Y 53.6187,Z 156,A 23.7181,B 16.1477,C -0.3386,E1 16.2961,E2 425.2764} C_DIS
LIN {X 115.7988,Y 56.4199,Z 156,A 25.0648,B 16.1476,C -0.3412,E1 16.2945,E2 423.9321} C_DIS
LIN {X 114.2974,Y 59.4018,Z 156,A 26.6163,B 16.1475,C -0.3474,E1 16.2925,E2 422.3714} C_DIS
LIN {X 112.6322,Y 62.5036,Z 156,A 28.1236,B 16.1475,C -0.3495,E1 16.2905,E2 420.8696} C_DIS
LIN {X 111.0658,Y 65.2463,Z 156,A 29.4101,B 16.1475,C -0.3489,E1 16.2887,E2 419.5957} C_DIS
LIN {X 109.6699,Y 67.5667,Z 156,A 30.7783,B 16.1472,C -0.3577,E1 16.2867,E2 418.2074} C_DIS
LIN {X 107.3777,Y 71.1537,Z 156,A 32.6868,B 16.1472,C -0.3629,E1 16.2838,E2 416.2956} C_DIS
LIN {X 105.152,Y 74.4028,Z 156,A 34.4252,B 16.147,C -0.3667,E1 16.281,E2 414.5574} C_DIS
LIN {X 102.784,Y 77.641,Z 156,A 36.1709,B 16.147,C -0.3696,E1 16.2781,E2 412.8148} C_DIS
LIN {X 100.4311,Y 80.6619,Z 156,A 37.9046,B 16.1469,C -0.3746,E1 16.2751,E2 411.0763} C_DIS
LIN {X 97.6831,Y 83.9685,Z 156,A 39.7717,B 16.1469,C -0.3773,E1 16.2717,E2 409.2132} C_DIS
LIN {X 94.9157,Y 87.0845,Z 156,A 41.6292,B 16.1467,C -0.3815,E1 16.2682,E2 407.3541} C_DIS
LIN {X 92.0501,Y 90.1081,Z 156,A 43.4731,B 16.1467,C -0.3851,E1 16.2647,E2 405.5101} C_DIS
LIN {X 88.8233,Y 93.2907,Z 156,A 45.4909,B 16.1465,C -0.3893,E1 16.2606,E2 403.4911} C_DIS
LIN {X 85.914,Y 95.9764,Z 156,A 47.2239,B 16.1465,C -0.3918,E1 16.257,E2 401.7604} C_DIS
LIN {X 82.5034,Y 98.9242,Z 156,A 49.1638,B 16.1465,C -0.3933,E1 16.2529,E2 399.8271} C_DIS
LIN {X 79.4117,Y 101.4224,Z 156,A 50.9067,B 16.1464,C -0.3956,E1 16.2491,E2 398.0864} C_DIS
LIN {X 76.1385,Y 103.902,Z 156,A 52.7563,B 16.1463,C -0.3996,E1 16.245,E2 396.2334} C_DIS
LIN {X 72.8778,Y 106.2144,Z 156,A 54.5316,B 16.1463,C -0.4024,E1 16.2409,E2 394.4578} C_DIS
LIN {X 69.8767,Y 108.2129,Z 156,A 56.1308,B 16.1462,C -0.4048,E1 16.2372,E2 392.8587} C_DIS
LIN {X 66.2693,Y 110.4591,Z 156,A 57.9286,B 16.1462,C -0.4045,E1 16.2329,E2 391.071} C_DIS
LIN {X 63.6338,Y 111.9976,Z 156,A 59.3125,B 16.1461,C -0.4073,E1 16.2295,E2 389.6838} C_DIS
LIN {X 60.7226,Y 113.6025,Z 156,A 60.8752,B 16.146,C -0.4121,E1 16.2257,E2 388.1111} C_DIS
LIN {X 57.5182,Y 115.257,Z 156,A 62.3477,B 16.146,C -0.4098,E1 16.2221,E2 386.6535} C_DIS
LIN {X 54.6798,Y 116.6309,Z 156,A 63.9291,B 16.1458,C -0.4174,E1 16.218,E2 385.0513} C_DIS
LIN {X 51.758,Y 117.9567,Z 156,A 65.2896,B 16.1458,C -0.4168,E1 16.2146,E2 383.6984} C_DIS
LIN {X 48.9363,Y 119.1554,Z 156,A 66.5382,B 16.1459,C -0.4144,E1 16.2114,E2 382.463} C_DIS
LIN {X 46.1264,Y 120.2701,Z 156,A 67.867,B 16.1459,C -0.4153,E1 16.2079,E2 381.136} C_DIS
LIN {X 43.51,Y 121.24,Z 156,A 69.1289,B 16.1459,C -0.4171,E1 16.2046,E2 379.8717} C_DIS
LIN {X 40.4085,Y 122.3089,Z 156,A 70.5813,B 16.1459,C -0.4182,E1 16.2008,E2 378.4202} C_DIS
LIN {X 37.3918,Y 123.2647,Z 156,A 72.0355,B 16.1458,C -0.4208,E1 16.1969,E2 376.9607} C_DIS
LIN {X 33.919,Y 124.2671,Z 156,A 73.61,B 16.1458,C -0.4208,E1 16.1926,E2 375.3902} C_DIS
LIN {X 30.2039,Y 125.2197,Z 156,A 75.0413,B 16.146,C -0.413,E1 16.1889,E2 373.9907} C_DIS
LIN {X 27.7975,Y 125.7774,Z 156,A 76.3102,B 16.1458,C -0.4191,E1 16.1853,E2 372.7025} C_DIS
LIN {X 24.7107,Y 126.4196,Z 156,A 77.6722,B 16.1458,C -0.4185,E1 16.1816,E2 371.3455} C_DIS
LIN {X 21.5678,Y 126.993,Z 156,A 79.1963,B 16.1458,C -0.4225,E1 16.1774,E2 369.8099} C_DIS
LIN {X 18.4668,Y 127.4806,Z 156,A 80.4402,B 16.1458,C -0.418,E1 16.174,E2 368.5838} C_DIS
LIN {X 15.3559,Y 127.8925,Z 156,A 82.0758,B 16.1456,C -0.4262,E1 16.1694,E2 366.9211} C_DIS
LIN {X 11.1084,Y 128.3315,Z 156,A 83.8807,B 16.1456,C -0.4235,E1 16.1644,E2 365.1278} C_DIS
LIN {X 7.0849,Y 128.6176,Z 156,A 85.8882,B 16.1456,C -0.4305,E1 16.1588,E2 363.0966} C_DIS
LIN {X 3.0884,Y 128.7751,Z 156,A 87.4008,B 16.1457,C -0.4219,E1 16.1546,E2 361.6153} C_DIS
LIN {X 0.002,Y 128.8132,Z 156,A 88.8516,B 16.1457,C -0.4243,E1 16.1506,E2 360.1563} C_DIS
LIN {X -3.1583,Y 128.7731,Z 156,A 90.2469,B 16.1457,C -0.4237,E1 16.1467,E2 358.7629} C_DIS
LIN {X -7.2537,Y 128.6085,Z 156,A 92.2278,B 16.1456,C -0.4283,E1 16.1411,E2 356.7648} C_DIS
LIN {X -11.0968,Y 128.3325,Z 156,A 93.8297,B 16.1456,C -0.4241,E1 16.1367,E2 355.1767} C_DIS
LIN {X -15.3475,Y 127.8935,Z 156,A 95.7291,B 16.1457,C -0.4233,E1 16.1314,E2 353.2786} C_DIS
LIN {X -18.9056,Y 127.4179,Z 156,A 97.2667,B 16.1457,C -0.4205,E1 16.1272,E2 351.7489} C_DIS
LIN {X -22.4496,Y 126.8398,Z 156,A 98.7264,B 16.1459,C -0.4153,E1 16.1232,E2 350.306} C_DIS
LIN {X -25.5372,Y 126.2542,Z 156,A 100.1396,B 16.1459,C -0.4148,E1 16.1193,E2 348.892} C_DIS
LIN {X -28.2187,Y 125.6828,Z 156,A 101.506,B 16.1459,C -0.4184,E1 16.1156,E2 347.5098} C_DIS
LIN {X -31.302,Y 124.9503,Z 156,A 102.9181,B 16.1459,C -0.4174,E1 16.1117,E2 346.0985} C_DIS
LIN {X -34.354,Y 124.1457,Z 156,A 104.325,B 16.1459,C -0.4162,E1 16.1079,E2 344.6924} C_DIS
LIN {X -37.8118,Y 123.1361,Z 156,A 105.9985,B 16.1459,C -0.4168,E1 16.1034,E2 343.012} C_DIS
LIN {X -41.8893,Y 121.8097,Z 156,A 107.8489,B 16.1459,C -0.4131,E1 16.0986,E2 341.1698} C_DIS
LIN {X -44.88,Y 120.7398,Z 156,A 109.2618,B 16.1459,C -0.4114,E1 16.0949,E2 339.7582} C_DIS
LIN {X -47.8287,Y 119.6024,Z 156,A 110.6763,B 16.146,C -0.41,E1 16.0912,E2 338.3439} C_DIS
LIN {X -50.7587,Y 118.3887,Z 156,A 112.0871,B 16.146,C -0.4082,E1 16.0876,E2 336.9344} C_DIS
LIN {X -53.6437,Y 117.11,Z 156,A 113.4954,B 16.1461,C -0.4065,E1 16.084,E2 335.527} C_DIS
LIN {X -56.4963,Y 115.7611,Z 156,A 114.9033,B 16.1461,C -0.4046,E1 16.0804,E2 334.12} C_DIS
LIN {X -59.7098,Y 114.1357,Z 156,A 116.4546,B 16.1463,C -0.4007,E1 16.0766,E2 332.5761} C_DIS
LIN {X -62.4817,Y 112.6442,Z 156,A 117.9276,B 16.1463,C -0.4007,E1 16.073,E2 331.0963} C_DIS
LIN {X -65.2455,Y 111.0662,Z 156,A 119.3694,B 16.1463,C -0.3992,E1 16.0695,E2 329.653} C_DIS
LIN {X -68.5424,Y 109.0627,Z 156,A 121.1697,B 16.1463,C -0.3989,E1 16.0652,E2 327.8449} C_DIS
LIN {X -71.5685,Y 107.1011,Z 156,A 122.764,B 16.1463,C -0.3957,E1 16.0615,E2 326.2535} C_DIS
LIN {X -74.5371,Y 105.0573,Z 156,A 124.448,B 16.1463,C -0.3952,E1 16.0576,E2 324.5621} C_DIS
LIN {X -77.9932,Y 102.5175,Z 156,A 126.3448,B 16.1465,C -0.3913,E1 16.0534,E2 322.6687} C_DIS
LIN {X -81.1085,Y 100.0709,Z 156,A 128.0345,B 16.1466,C -0.3856,E1 16.0497,E2 320.9894} C_DIS
LIN {X -84.3055,Y 97.3929,Z 156,A 129.9848,B 16.1466,C -0.3846,E1 16.0455,E2 319.0304} C_DIS
Enddeposition()
END
